ABB RAPID module: TaskModule.mod

MODULE TaskModule
    !*****************************************************
    !Module Name: TaskModule
    !Version:     1.0
    !Description: This module stroes ths data which are not shared among other tasks
    !Date:        2018-8-10
    !Author:      Michael
    !*****************************************************

    VAR num numStation:=1;
    VAR partdata pdTmpChk;
    VAR string sPartDataName;

    CONST num numPedestalBottomWidth:=100;
    CONST num numPedestalBottomHeight:=505;
    CONST num numPedestalAngle:=90;
    PERS num numPedestalVertexHeight:=455;

    VAR syncident SyncPositionerHomed;
    VAR syncident SyncWobjScanning;
    VAR syncident SyncWobjBranchScaning;
    VAR syncident SyncWobjBranchScaned;
    VAR syncident SyncWobjHeaderScaning;
    VAR syncident SyncWobjHeaderScaned;
    VAR syncident SyncWobjBranchScaningV2;
    VAR syncident SyncWobjBranchScanedV2;
    VAR syncident SyncWobjHeaderScaningV2;
    VAR syncident SyncWobjHeaderScanedV2;
    VAR syncident SyncWobjScaned;
    VAR syncident SyncBranchPeripherySmarTac;
    VAR syncident SyncHeaderPeripherySmarTac;
    VAR syncident SyncWobjRevised;

    VAR syncident SyncPositionerWeldApproached;
    VAR syncident SyncRobotsWeldApproached;
    VAR syncident SyncAllRobotsWeldStart;
    VAR syncident SyncAllRobotsWeldEnd;
    VAR syncident SyncRobotsWeldDeparted;

    VAR syncident SyncMoveLSubstituted1;
    VAR syncident SyncMoveLSubstituted2;

    VAR syncident SyncRobotsForTest11;
    VAR syncident SyncRobotsForTest12;
    VAR syncident SyncRobotsForTest13;

    VAR syncident SyncRobotsForTest21;
    VAR syncident SyncRobotsForTest22;
    VAR syncident SyncRobotsForTest23;
    VAR syncident SyncRobotsForTest24;
    VAR syncident SyncRobotsForTest25;
    VAR syncident SyncRobotsForTest26;

    VAR syncident SyncVerifyTrackHorizontal1;
    VAR syncident SyncVerifyTrackHorizontal2;
    VAR syncident SyncVerifyTrackHorizontal3;
    VAR syncident SyncVerifyTrackHorizontal4;
    VAR syncident SyncVerifyTrackHorizontal5;
    VAR syncident SyncVerifyTrackHorizontal6;
    VAR syncident SyncVerifyTrackHorizontal7;
    VAR syncident SyncVerifyTrackHorizontal8;

    VAR string strCurTaskName:="T_ROB1";
    VAR num numCurTaskNo:=1;
    VAR num numRobLayerCurTotal;
    VAR RECORDWeldTarget rRobLayerCur{30};
    VAR RECORDLayerParamter rLayerParamterCur;

    TASK PERS tooldata toolWeldGun:=[TRUE,[[80.8801,-0.792657,372.832],[0.950301,0.00218631,0.311128,-0.0110736]],[5.2,[34.6,-12.3,73.3],[1,0,0,0],0.048,0.077,0.012]];
    TASK PERS tooldata toolLaser:=[TRUE,[[-54.9581,16.2889,420.256],[0.999173,0.00179167,-0.00748378,0.0399198]],[5.2,[34.6,-12.3,73.3],[1,0,0,0],0.048,0.077,0.012]];
    TASK PERS extjoint extjointValue:=[4816.37,9E+09,9E+09,9E+09,9E+09,9E+09];

    TASK PERS robtarget robtApproachPlatoonSinking:=[[380,-200,190.17],[0.0294666,-0.614745,0.74898,0.245457],[-1,-1,0,1],[4837,9E+09,9E+09,9E+09,9E+09,9E+09]];
    TASK PERS robtarget robtDepartPlatoonSinking:=[[380,-200,190.17],[0.0294677,-0.614743,0.748982,0.245457],[-1,-1,0,1],[4837,9E+09,9E+09,9E+09,9E+09,9E+09]];

    TASK PERS robtarget robtApproachSaddle:=[[487.15,-501.33,347.1],[0.31599,-0.0842611,-0.937489,-0.119018],[-1,0,0,0],[4837,9E+09,9E+09,9E+09,9E+09,9E+09]];
    TASK PERS robtarget robtDepartSaddle:=[[487.15,-501.33,347.1],[0.315989,-0.0842597,-0.937489,-0.119018],[-1,0,0,0],[4837,9E+09,9E+09,9E+09,9E+09,9E+09]];

    TASK PERS robtarget robtApproachSaddleScan:=[[380,-301.92,219.63],[0.442137,-0.896947,4.32324E-05,3.41344E-05],[-1,-1,-1,1],[4837,9E+09,9E+09,9E+09,9E+09,9E+09]];
    TASK PERS robtarget robtDepartSaddleScan:=[[380,-301.92,219.64],[0.442138,-0.896947,4.317E-05,3.4008E-05],[-1,-1,-1,1],[4837,9E+09,9E+09,9E+09,9E+09,9E+09]];

    TASK PERS robtarget robtApproachPlatoonSinkingScan:=[[380,238.1,333.7],[0.270598,0.653281,-0.653282,0.270598],[0,0,1,1],[4837,9E+09,9E+09,9E+09,9E+09,9E+09]];
    TASK PERS robtarget robtDepartPlatoonSinkingScan:=[[380,238.1,333.7],[0.270598,0.653281,-0.653282,0.270598],[0,0,1,1],[4837,9E+09,9E+09,9E+09,9E+09,9E+09]];

    TASK PERS confdata confPlatoonSinkingOrigin:=[0,0,-1,1];
    TASK PERS confdata confSaddleOrigin:=[-1,0,-1,0];

    TASK PERS robtarget robtNext:=[[149.55,3.75943E-07,159.914],[0.348789,0.457656,-0.792683,-0.201373],[-1,0,-1,0],[4217,9E+09,9E+09,9E+09,9E+09,9E+09]];
    TASK PERS robtarget robtCircleEnd:=[[149.55,3.75943E-07,159.914],[0.348789,0.457656,-0.792683,-0.201373],[-1,1,-2,0],[4217,9E+09,9E+09,9E+09,9E+09,9E+09]];

    TASK PERS seamdata seamNext:=[0,0.5,[0,0,0,100,0,0,0,0,0],0,0,5,0,0,[0,0,1,140,0,0,0,0,0],0,1.5,[0,0,1,90,0,0,0,0,0],0.04,0,[0,0,0,0,0,0,0,0,0],0.5];
    TASK PERS welddata weldNext:=[7,0,[47,0,0,0,0,240,0,0,0],[0,0,0,0,0,0,0,0,0]];
    TASK PERS weavedata weaveNext:=[1,0,3.5,0,0,0,0,0,0,0,0,0,0,0,0];
    TASK PERS trackdata trackNext:=[0,FALSE,50,[0,0,0,0,0,0,0,0,0],[0,0,0,0,0,0,0]];
    TASK PERS adaptdata adaptNext:=[0,1,0,0,0.1,100,0.1,100];
    TASK PERS num numWeaveWidth90:=0;
    TASK PERS num numGrooveWidthNext:=0;

    VAR clock clockPartTimeConsume;
    TASK PERS num numTimeConsumeTotal:=623.885;

    !numTCSRotationX
    TASK PERS num numPlatoonSinkingPushDragAngle:=45;
    !numTCSRotationY
    TASK PERS num numPlatoonSinkingWorkAngle:=-10;

    TASK PERS jointtarget jointNext:=[[9E+09,9E+09,9E+09,9E+09,9E+09,9E+09],[0,66.4272,9E+09,9E+09,9E+09,9E+09]];
    TASK PERS speeddata speedLinearScan:=[19,500,5000,1000];

    TASK PERS string strWeldParametersLogFileName:="WeldParametersLog.csv";
    CONST string strWeldProcedureLogLogFileName:="WeldProcedureLog1.csv";

    CONST string strSSBLogFileName:="ScanSaddleBranch1.csv";
    CONST string strSSHLogFileName:="ScanSaddleHeader1.csv";

    !For saddle branch SmarTac
    TASK PERS num numSSBPointsTotal:=13;
    !Scan saddle branch range
    TASK PERS num numSSBAngleFrom:=225;
    TASK PERS num numSSBAngleTo:=330;

    !For saddle header SmarTac
    TASK PERS num numSSHPointsTotal:=13;
    !Scan saddle header range
    TASK PERS num numSSHAngleFrom:=180;
    TASK PERS num numSSHAngleTo:=90;

    !Scan saddle branch points
    TASK PERS robtarget robtSSBLaserSmarTacs{20}:=[[[339.589,-40.4111,208.15],[0.270598,0.270598,0.653282,0.653281],[0,0,0,1],[4837,9E+09,9E+09,9E+09,9E+09,9E+09]],[[346.207,-46.0883,208.15],[0.219975,0.219975,0.67202,0.67202],[0,0,0,1],[4837,9E+09,9E+09,9E+09,9E+09,9E+09]],[[353.611,-50.6927,208.15],[0.168069,0.168069,0.686843,0.686843],[0,0,0,1],[4837,9E+09,9E+09,9E+09,9E+09,9E+09]],[[361.63,-54.1171,208.15],[0.115184,0.115184,0.697662,0.697662],[0,0,0,1],[4837,9E+09,9E+09,9E+09,9E+09,9E+09]],[[370.076,-56.2818,208.15],[0.0616285,0.0616285,0.704416,0.704416],[0,0,0,1],[4837,9E+09,9E+09,9E+09,9E+09,9E+09]],[[378.753,-57.1364,208.15],[0.00771319,0.0077132,0.707065,0.707065],[0,0,1,1],[4837,9E+09,9E+09,9E+09,9E+09,9E+09]],[[387.46,-56.6611,208.15],[0.046247,0.046247,-0.705593,-0.705593],[-1,-1,1,1],[4837,9E+09,9E+09,9E+09,9E+09,9E+09]],[[395.992,-54.8668,208.15],[0.0999376,0.0999376,-0.700009,-0.700009],[-1,-1,1,1],[4837,9E+09,9E+09,9E+09,9E+09,9E+09]],[[404.153,-51.7955,208.15],[0.153046,0.153046,-0.690346,-0.690346],[-1,-1,1,1],[4837,9E+09,9E+09,9E+09,9E+09,9E+09]],[[411.751,-47.5185,208.15],[0.205262,0.205262,-0.676659,-0.676659],[-1,-1,1,1],[4837,9E+09,9E+09,9E+09,9E+09,9E+09]],[[418.61,-42.1354,208.15],[0.256282,0.256282,-0.659029,-0.659029],[-1,-1,1,1],[4837,9E+09,9E+09,9E+09,9E+09,9E+09]],[[424.57,-35.7715,208.15],[0.305809,0.305809,-0.637559,-0.637559],[-1,-1,1,1],[4837,9E+09,9E+09,9E+09,9E+09,9E+09]],[[429.493,-28.575,208.15],[0.353553,0.353553,-0.612372,-0.612372],[-1,-1,1,1],[4837,9E+09,9E+09,9E+09,9E+09,9E+09]],[[652.53,-493.33,1047.99],[0.459259,-0.544323,-0.447932,-0.54051],[-1,-1,1,1],[4837,9E+09,9E+09,9E+09,9E+09,9E+09]],[[652.53,-493.33,1047.99],[0.459259,-0.544323,-0.447932,-0.54051],[-1,0,-2,1],[4837,9E+09,9E+09,9E+09,9E+09,9E+09]],[[652.53,-493.33,1047.99],[0.459259,-0.544323,-0.447932,-0.54051],[-1,0,-2,1],[4837,9E+09,9E+09,9E+09,9E+09,9E+09]],[[652.53,-493.33,1047.99],[0.459259,-0.544323,-0.447932,-0.54051],[-1,0,-2,1],[4837,9E+09,9E+09,9E+09,9E+09,9E+09]],[[652.53,-493.33,1047.99],[0.459259,-0.544323,-0.447932,-0.54051],[-1,0,-2,1],[4837,9E+09,9E+09,9E+09,9E+09,9E+09]],[[652.53,-493.33,1047.99],[0.459259,-0.544323,-0.447932,-0.54051],[-1,0,-2,1],[4837,9E+09,9E+09,9E+09,9E+09,9E+09]],[[652.53,-493.33,1047.99],[0.459259,-0.544323,-0.447932,-0.54051],[-1,0,-2,1],[4837,9E+09,9E+09,9E+09,9E+09,9E+09]]];
    TASK PERS robtarget robtSSBWireSmarTacs{20}:=[[[428.493,28.575,188.15],[0.683013,0.183013,-0.683013,0.183013],[0,1,-3,1],[4838,9E+09,9E+09,9E+09,9E+09,9E+09]],[[422.779,36.7353,188.15],[0.664463,0.241845,-0.664463,0.241845],[0,1,-3,1],[4838,9E+09,9E+09,9E+09,9E+09,9E+09]],[[415.735,43.7794,188.15],[0.640856,0.298836,-0.640856,0.298836],[0,1,-3,1],[4838,9E+09,9E+09,9E+09,9E+09,9E+09]],[[407.575,49.4934,188.15],[0.612372,0.353553,-0.612372,0.353553],[0,0,-3,1],[4838,9E+09,9E+09,9E+09,9E+09,9E+09]],[[398.546,53.7034,188.15],[0.579228,0.40558,-0.579228,0.40558],[0,0,-3,1],[4838,9E+09,9E+09,9E+09,9E+09,9E+09]],[[388.924,56.2818,188.15],[0.541675,0.454519,-0.541675,0.454519],[0,0,-3,1],[4838,9E+09,9E+09,9E+09,9E+09,9E+09]],[[379,57.15,188.15],[0.5,0.5,-0.5,0.5],[0,0,-3,1],[4838,9E+09,9E+09,9E+09,9E+09,9E+09]],[[369.076,56.2818,188.15],[0.454519,0.541675,-0.454519,0.541675],[-1,-1,-2,1],[4838,9E+09,9E+09,9E+09,9E+09,9E+09]],[[359.454,53.7034,188.15],[0.40558,0.579228,-0.40558,0.579228],[-1,-1,-2,1],[4838,9E+09,9E+09,9E+09,9E+09,9E+09]],[[350.425,49.4934,188.15],[0.353553,0.612372,-0.353553,0.612372],[-1,-1,-2,1],[4838,9E+09,9E+09,9E+09,9E+09,9E+09]],[[342.265,43.7794,188.15],[0.298836,0.640856,-0.298836,0.640856],[-1,-2,-2,1],[4838,9E+09,9E+09,9E+09,9E+09,9E+09]],[[335.221,36.7353,188.15],[0.241845,0.664463,-0.241845,0.664463],[-1,-2,-2,1],[4838,9E+09,9E+09,9E+09,9E+09,9E+09]],[[329.507,28.575,188.15],[0.183013,0.683013,-0.183013,0.683013],[-1,-2,-2,1],[4838,9E+09,9E+09,9E+09,9E+09,9E+09]],[[652.53,-493.33,1047.99],[0.459259,-0.544323,-0.447932,-0.54051],[-1,-1,-2,1],[4837,9E+09,9E+09,9E+09,9E+09,9E+09]],[[652.53,-493.33,1047.99],[0.459259,-0.544323,-0.447932,-0.54051],[-1,0,-2,1],[4837,9E+09,9E+09,9E+09,9E+09,9E+09]],[[652.53,-493.33,1047.99],[0.459259,-0.544323,-0.447932,-0.54051],[-1,0,-2,1],[4837,9E+09,9E+09,9E+09,9E+09,9E+09]],[[652.53,-493.33,1047.99],[0.459259,-0.544323,-0.447932,-0.54051],[-1,0,-2,1],[4837,9E+09,9E+09,9E+09,9E+09,9E+09]],[[652.53,-493.33,1047.99],[0.459259,-0.544323,-0.447932,-0.54051],[-1,0,-2,1],[4837,9E+09,9E+09,9E+09,9E+09,9E+09]],[[652.53,-493.33,1047.99],[0.459259,-0.544323,-0.447932,-0.54051],[-1,0,-2,1],[4837,9E+09,9E+09,9E+09,9E+09,9E+09]],[[652.53,-493.33,1047.99],[0.459259,-0.544323,-0.447932,-0.54051],[-1,0,-2,1],[4837,9E+09,9E+09,9E+09,9E+09,9E+09]]];
    TASK PERS robtarget robtSSBLinerFrom:=[[427.815,-90,208.15],[3.09086E-08,3.09086E-08,-0.707107,-0.707107],[0,0,1,1],[4837,9E+09,9E+09,9E+09,9E+09,9E+09]];
    TASK PERS robtarget robtSSBLinerTo:=[[427.815,-90,208.15],[3.09086E-08,3.09086E-08,-0.707107,-0.707107],[0,0,1,1],[4837,9E+09,9E+09,9E+09,9E+09,9E+09]];

    !Scan saddle branch results, shared for all the four scan methods
    TASK PERS pose poseSSBs{20}:=[[[17.952,17.949,-0.0153198],[1,0,0,0]],[[1.39819,1.89476,-0.013504],[1,0,0,0]],[[1.19794,2.30891,-0.0127716],[1,0,0,0]],[[1.09225,3.15936,0.00701904],[1,0,0,0]],[[0.711761,4.05244,0.0107269],[1,0,0,0]],[[0.0821533,3.84193,-0.0236664],[1,0,0,0]],[[-0.370331,2.84446,0.0133057],[1,0,0,0]],[[-0.622101,2.14712,0.00906372],[1,0,0,0]],[[-1.77264,3.79015,0.0375366],[1,0,0,0]],[[-2.026,3.00191,-0.0130768],[1,0,0,0]],[[-5.25485,5.71828,0.0316315],[1,0,0,0]],[[-2.63602,2.12254,-0.0143127],[1,0,0,0]],[[-2.9296,1.71353,0.0193481],[1,0,0,0]],[[0,0,0],[1,0,0,0]],[[0,0,0],[1,0,0,0]],[[0,0,0],[1,0,0,0]],[[0,0,0],[1,0,0,0]],[[0,0,0],[1,0,0,0]],[[0,0,0],[1,0,0,0]],[[0,0,0],[1,0,0,0]]];
    TASK PERS num numSSBLaserValues{100}:=[0,0,0,0,0,0,0,0,0,0,0,0,0,0,0,0,0,0,0,0,0,0,0,0,0,0,0,0,0,0,0,0,0,0,0,0,0,0,0,0,0,0,0,0,0,0,0,0,0,0,0,0,0,0,0,0,0,0,0,0,0,0,0,0,0,0,0,0,0,0,0,0,0,0,0,0,0,0,0,0,0,0,0,0,0,0,0,0,0,0,0,0,0,0,0,0,0,0,0,0];
    TASK PERS robtarget robtSSBPeripherys{100}:=[[[920.345,-94.6578,259.235],[0.270602,0.270593,0.653289,0.653275],[0,0,0,1],[4202,9E+09,9E+09,9E+09,9E+09,9E+09]],[[347.605,-44.1936,208.136],[0.219979,0.219977,0.672024,0.672014],[0,0,0,1],[4837,9E+09,9E+09,9E+09,9E+09,9E+09]],[[354.809,-48.3838,208.137],[0.168074,0.168066,0.686843,0.686841],[0,0,0,1],[4837,9E+09,9E+09,9E+09,9E+09,9E+09]],[[362.722,-50.9577,208.157],[0.115179,0.115206,0.697653,0.697669],[0,0,0,1],[4837,9E+09,9E+09,9E+09,9E+09,9E+09]],[[370.788,-52.2293,208.161],[0.0616358,0.0616132,0.704405,0.704427],[0,0,0,1],[4837,9E+09,9E+09,9E+09,9E+09,9E+09]],[[378.835,-53.2945,208.126],[0.00771569,0.00771062,0.707077,0.707053],[0,0,1,1],[4837,9E+09,9E+09,9E+09,9E+09,9E+09]],[[387.089,-53.8166,208.163],[0.0462415,0.0462523,-0.705592,-0.705594],[-1,-1,1,1],[4837,9E+09,9E+09,9E+09,9E+09,9E+09]],[[395.37,-52.7197,208.159],[0.0999338,0.0999283,-0.700005,-0.700014],[-1,-1,1,1],[4837,9E+09,9E+09,9E+09,9E+09,9E+09]],[[402.38,-48.0053,208.188],[0.153049,0.153049,-0.690324,-0.690366],[-1,-1,1,1],[4837,9E+09,9E+09,9E+09,9E+09,9E+09]],[[409.725,-44.5166,208.137],[0.205273,0.20527,-0.676661,-0.676652],[-1,-1,1,1],[4837,9E+09,9E+09,9E+09,9E+09,9E+09]],[[413.355,-36.4171,208.182],[0.256285,0.256298,-0.659006,-0.659045],[-1,-1,1,1],[4837,9E+09,9E+09,9E+09,9E+09,9E+09]],[[421.934,-33.649,208.136],[0.305815,0.3058,-0.637569,-0.637549],[-1,-1,1,1],[4837,9E+09,9E+09,9E+09,9E+09,9E+09]],[[426.564,-26.8615,208.169],[0.353544,0.353553,-0.612368,-0.612383],[-1,-1,1,1],[4837,9E+09,9E+09,9E+09,9E+09,9E+09]],[[75.54,-110.49,75.53],[0.104911,-0.592891,0.59209,0.535634],[-1,-2,0,1],[3747.5,9E+09,9E+09,9E+09,9E+09,9E+09]],[[75.54,-110.49,75.53],[0.104911,-0.592891,0.59209,0.535634],[-1,0,-1,0],[3747.5,9E+09,9E+09,9E+09,9E+09,9E+09]],[[75.54,-110.49,75.53],[0.104911,-0.592891,0.59209,0.535634],[-1,0,-1,0],[3747.5,9E+09,9E+09,9E+09,9E+09,9E+09]],[[75.54,-110.49,75.53],[0.104911,-0.592891,0.59209,0.535634],[-1,0,-1,0],[3747.5,9E+09,9E+09,9E+09,9E+09,9E+09]],[[75.54,-110.49,75.53],[0.104911,-0.592891,0.59209,0.535634],[-1,0,-1,0],[3747.5,9E+09,9E+09,9E+09,9E+09,9E+09]],[[75.54,-110.49,75.53],[0.104911,-0.592891,0.59209,0.535634],[-1,0,-1,0],[3747.5,9E+09,9E+09,9E+09,9E+09,9E+09]],[[75.54,-110.49,75.53],[0.104911,-0.592891,0.59209,0.535634],[-1,0,-1,0],[3747.5,9E+09,9E+09,9E+09,9E+09,9E+09]],[[75.54,-110.49,75.53],[0.104911,-0.592891,0.59209,0.535634],[-1,0,-1,0],[3747.5,9E+09,9E+09,9E+09,9E+09,9E+09]],[[75.54,-110.49,75.53],[0.104911,-0.592891,0.59209,0.535634],[-1,0,-1,0],[3747.5,9E+09,9E+09,9E+09,9E+09,9E+09]],[[75.54,-110.49,75.53],[0.104911,-0.592891,0.59209,0.535634],[-1,0,-1,0],[3747.5,9E+09,9E+09,9E+09,9E+09,9E+09]],[[75.54,-110.49,75.53],[0.104911,-0.592891,0.59209,0.535634],[-1,0,-1,0],[3747.5,9E+09,9E+09,9E+09,9E+09,9E+09]],[[75.54,-110.49,75.53],[0.104911,-0.592891,0.59209,0.535634],[-1,0,-1,0],[3747.5,9E+09,9E+09,9E+09,9E+09,9E+09]],[[75.54,-110.49,75.53],[0.104911,-0.592891,0.59209,0.535634],[-1,0,-1,0],[3747.5,9E+09,9E+09,9E+09,9E+09,9E+09]],[[75.54,-110.49,75.53],[0.104911,-0.592891,0.59209,0.535634],[-1,0,-1,0],[3747.5,9E+09,9E+09,9E+09,9E+09,9E+09]],[[75.54,-110.49,75.53],[0.104911,-0.592891,0.59209,0.535634],[-1,0,-1,0],[3747.5,9E+09,9E+09,9E+09,9E+09,9E+09]],[[75.54,-110.49,75.53],[0.104911,-0.592891,0.59209,0.535634],[-1,0,-1,0],[3747.5,9E+09,9E+09,9E+09,9E+09,9E+09]],[[75.54,-110.49,75.53],[0.104911,-0.592891,0.59209,0.535634],[-1,0,-1,0],[3747.5,9E+09,9E+09,9E+09,9E+09,9E+09]],[[75.54,-110.49,75.53],[0.104911,-0.592891,0.59209,0.535634],[-1,0,-1,0],[3747.5,9E+09,9E+09,9E+09,9E+09,9E+09]],[[75.54,-110.49,75.53],[0.104911,-0.592891,0.59209,0.535634],[-1,0,-1,0],[3747.5,9E+09,9E+09,9E+09,9E+09,9E+09]],[[75.54,-110.49,75.53],[0.104911,-0.592891,0.59209,0.535634],[-1,0,-1,0],[3747.5,9E+09,9E+09,9E+09,9E+09,9E+09]],[[75.54,-110.49,75.53],[0.104911,-0.592891,0.59209,0.535634],[-1,0,-1,0],[3747.5,9E+09,9E+09,9E+09,9E+09,9E+09]],[[75.54,-110.49,75.53],[0.104911,-0.592891,0.59209,0.535634],[-1,0,-1,0],[3747.5,9E+09,9E+09,9E+09,9E+09,9E+09]],[[75.54,-110.49,75.53],[0.104911,-0.592891,0.59209,0.535634],[-1,0,-1,0],[3747.5,9E+09,9E+09,9E+09,9E+09,9E+09]],[[75.54,-110.49,75.53],[0.104911,-0.592891,0.59209,0.535634],[-1,0,-1,0],[3747.5,9E+09,9E+09,9E+09,9E+09,9E+09]],[[75.54,-110.49,75.53],[0.104911,-0.592891,0.59209,0.535634],[-1,0,-1,0],[3747.5,9E+09,9E+09,9E+09,9E+09,9E+09]],[[75.54,-110.49,75.53],[0.104911,-0.592891,0.59209,0.535634],[-1,0,-1,0],[3747.5,9E+09,9E+09,9E+09,9E+09,9E+09]],[[75.54,-110.49,75.53],[0.104911,-0.592891,0.59209,0.535634],[-1,0,-1,0],[3747.5,9E+09,9E+09,9E+09,9E+09,9E+09]],[[75.54,-110.49,75.53],[0.104911,-0.592891,0.59209,0.535634],[-1,0,-1,0],[3747.5,9E+09,9E+09,9E+09,9E+09,9E+09]],[[75.54,-110.49,75.53],[0.104911,-0.592891,0.59209,0.535634],[-1,0,-1,0],[3747.5,9E+09,9E+09,9E+09,9E+09,9E+09]],[[75.54,-110.49,75.53],[0.104911,-0.592891,0.59209,0.535634],[-1,0,-1,0],[3747.5,9E+09,9E+09,9E+09,9E+09,9E+09]],[[75.54,-110.49,75.53],[0.104911,-0.592891,0.59209,0.535634],[-1,0,-1,0],[3747.5,9E+09,9E+09,9E+09,9E+09,9E+09]],[[75.54,-110.49,75.53],[0.104911,-0.592891,0.59209,0.535634],[-1,0,-1,0],[3747.5,9E+09,9E+09,9E+09,9E+09,9E+09]],[[75.54,-110.49,75.53],[0.104911,-0.592891,0.59209,0.535634],[-1,0,-1,0],[3747.5,9E+09,9E+09,9E+09,9E+09,9E+09]],[[75.54,-110.49,75.53],[0.104911,-0.592891,0.59209,0.535634],[-1,0,-1,0],[3747.5,9E+09,9E+09,9E+09,9E+09,9E+09]],[[75.54,-110.49,75.53],[0.104911,-0.592891,0.59209,0.535634],[-1,0,-1,0],[3747.5,9E+09,9E+09,9E+09,9E+09,9E+09]],[[75.54,-110.49,75.53],[0.104911,-0.592891,0.59209,0.535634],[-1,0,-1,0],[3747.5,9E+09,9E+09,9E+09,9E+09,9E+09]],[[75.54,-110.49,75.53],[0.104911,-0.592891,0.59209,0.535634],[-1,0,-1,0],[3747.5,9E+09,9E+09,9E+09,9E+09,9E+09]],[[75.54,-110.49,75.53],[0.104911,-0.592891,0.59209,0.535634],[-1,0,-1,0],[3747.5,9E+09,9E+09,9E+09,9E+09,9E+09]],[[75.54,-110.49,75.53],[0.104911,-0.592891,0.59209,0.535634],[-1,0,-1,0],[3747.5,9E+09,9E+09,9E+09,9E+09,9E+09]],[[75.54,-110.49,75.53],[0.104911,-0.592891,0.59209,0.535634],[-1,0,-1,0],[3747.5,9E+09,9E+09,9E+09,9E+09,9E+09]],[[75.54,-110.49,75.53],[0.104911,-0.592891,0.59209,0.535634],[-1,0,-1,0],[3747.5,9E+09,9E+09,9E+09,9E+09,9E+09]],[[75.54,-110.49,75.53],[0.104911,-0.592891,0.59209,0.535634],[-1,0,-1,0],[3747.5,9E+09,9E+09,9E+09,9E+09,9E+09]],[[75.54,-110.49,75.53],[0.104911,-0.592891,0.59209,0.535634],[-1,0,-1,0],[3747.5,9E+09,9E+09,9E+09,9E+09,9E+09]],[[75.54,-110.49,75.53],[0.104911,-0.592891,0.59209,0.535634],[-1,0,-1,0],[3747.5,9E+09,9E+09,9E+09,9E+09,9E+09]],[[75.54,-110.49,75.53],[0.104911,-0.592891,0.59209,0.535634],[-1,0,-1,0],[3747.5,9E+09,9E+09,9E+09,9E+09,9E+09]],[[75.54,-110.49,75.53],[0.104911,-0.592891,0.59209,0.535634],[-1,0,-1,0],[3747.5,9E+09,9E+09,9E+09,9E+09,9E+09]],[[75.54,-110.49,75.53],[0.104911,-0.592891,0.59209,0.535634],[-1,0,-1,0],[3747.5,9E+09,9E+09,9E+09,9E+09,9E+09]],[[75.54,-110.49,75.53],[0.104911,-0.592891,0.59209,0.535634],[-1,0,-1,0],[3747.5,9E+09,9E+09,9E+09,9E+09,9E+09]],[[75.54,-110.49,75.53],[0.104911,-0.592891,0.59209,0.535634],[-1,0,-1,0],[3747.5,9E+09,9E+09,9E+09,9E+09,9E+09]],[[75.54,-110.49,75.53],[0.104911,-0.592891,0.59209,0.535634],[-1,0,-1,0],[3747.5,9E+09,9E+09,9E+09,9E+09,9E+09]],[[75.54,-110.49,75.53],[0.104911,-0.592891,0.59209,0.535634],[-1,0,-1,0],[3747.5,9E+09,9E+09,9E+09,9E+09,9E+09]],[[75.54,-110.49,75.53],[0.104911,-0.592891,0.59209,0.535634],[-1,0,-1,0],[3747.5,9E+09,9E+09,9E+09,9E+09,9E+09]],[[75.54,-110.49,75.53],[0.104911,-0.592891,0.59209,0.535634],[-1,0,-1,0],[3747.5,9E+09,9E+09,9E+09,9E+09,9E+09]],[[75.54,-110.49,75.53],[0.104911,-0.592891,0.59209,0.535634],[-1,0,-1,0],[3747.5,9E+09,9E+09,9E+09,9E+09,9E+09]],[[75.54,-110.49,75.53],[0.104911,-0.592891,0.59209,0.535634],[-1,0,-1,0],[3747.5,9E+09,9E+09,9E+09,9E+09,9E+09]],[[75.54,-110.49,75.53],[0.104911,-0.592891,0.59209,0.535634],[-1,0,-1,0],[3747.5,9E+09,9E+09,9E+09,9E+09,9E+09]],[[75.54,-110.49,75.53],[0.104911,-0.592891,0.59209,0.535634],[-1,0,-1,0],[3747.5,9E+09,9E+09,9E+09,9E+09,9E+09]],[[75.54,-110.49,75.53],[0.104911,-0.592891,0.59209,0.535634],[-1,0,-1,0],[3747.5,9E+09,9E+09,9E+09,9E+09,9E+09]],[[75.54,-110.49,75.53],[0.104911,-0.592891,0.59209,0.535634],[-1,0,-1,0],[3747.5,9E+09,9E+09,9E+09,9E+09,9E+09]],[[75.54,-110.49,75.53],[0.104911,-0.592891,0.59209,0.535634],[-1,0,-1,0],[3747.5,9E+09,9E+09,9E+09,9E+09,9E+09]],[[75.54,-110.49,75.53],[0.104911,-0.592891,0.59209,0.535634],[-1,0,-1,0],[3747.5,9E+09,9E+09,9E+09,9E+09,9E+09]],[[75.54,-110.49,75.53],[0.104911,-0.592891,0.59209,0.535634],[-1,0,-1,0],[3747.5,9E+09,9E+09,9E+09,9E+09,9E+09]],[[75.54,-110.49,75.53],[0.104911,-0.592891,0.59209,0.535634],[-1,0,-1,0],[3747.5,9E+09,9E+09,9E+09,9E+09,9E+09]],[[75.54,-110.49,75.53],[0.104911,-0.592891,0.59209,0.535634],[-1,0,-1,0],[3747.5,9E+09,9E+09,9E+09,9E+09,9E+09]],[[75.54,-110.49,75.53],[0.104911,-0.592891,0.59209,0.535634],[-1,0,-1,0],[3747.5,9E+09,9E+09,9E+09,9E+09,9E+09]],[[75.54,-110.49,75.53],[0.104911,-0.592891,0.59209,0.535634],[-1,0,-1,0],[3747.5,9E+09,9E+09,9E+09,9E+09,9E+09]],[[75.54,-110.49,75.53],[0.104911,-0.592891,0.59209,0.535634],[-1,0,-1,0],[3747.5,9E+09,9E+09,9E+09,9E+09,9E+09]],[[75.54,-110.49,75.53],[0.104911,-0.592891,0.59209,0.535634],[-1,0,-1,0],[3747.5,9E+09,9E+09,9E+09,9E+09,9E+09]],[[75.54,-110.49,75.53],[0.104911,-0.592891,0.59209,0.535634],[-1,0,-1,0],[3747.5,9E+09,9E+09,9E+09,9E+09,9E+09]],[[75.54,-110.49,75.53],[0.104911,-0.592891,0.59209,0.535634],[-1,0,-1,0],[3747.5,9E+09,9E+09,9E+09,9E+09,9E+09]],[[75.54,-110.49,75.53],[0.104911,-0.592891,0.59209,0.535634],[-1,0,-1,0],[3747.5,9E+09,9E+09,9E+09,9E+09,9E+09]],[[75.54,-110.49,75.53],[0.104911,-0.592891,0.59209,0.535634],[-1,0,-1,0],[3747.5,9E+09,9E+09,9E+09,9E+09,9E+09]],[[75.54,-110.49,75.53],[0.104911,-0.592891,0.59209,0.535634],[-1,0,-1,0],[3747.5,9E+09,9E+09,9E+09,9E+09,9E+09]],[[75.54,-110.49,75.53],[0.104911,-0.592891,0.59209,0.535634],[-1,0,-1,0],[3747.5,9E+09,9E+09,9E+09,9E+09,9E+09]],[[75.54,-110.49,75.53],[0.104911,-0.592891,0.59209,0.535634],[-1,0,-1,0],[3747.5,9E+09,9E+09,9E+09,9E+09,9E+09]],[[75.54,-110.49,75.53],[0.104911,-0.592891,0.59209,0.535634],[-1,0,-1,0],[3747.5,9E+09,9E+09,9E+09,9E+09,9E+09]],[[75.54,-110.49,75.53],[0.104911,-0.592891,0.59209,0.535634],[-1,0,-1,0],[3747.5,9E+09,9E+09,9E+09,9E+09,9E+09]],[[75.54,-110.49,75.53],[0.104911,-0.592891,0.59209,0.535634],[-1,0,-1,0],[3747.5,9E+09,9E+09,9E+09,9E+09,9E+09]],[[75.54,-110.49,75.53],[0.104911,-0.592891,0.59209,0.535634],[-1,0,-1,0],[3747.5,9E+09,9E+09,9E+09,9E+09,9E+09]],[[75.54,-110.49,75.53],[0.104911,-0.592891,0.59209,0.535634],[-1,0,-1,0],[3747.5,9E+09,9E+09,9E+09,9E+09,9E+09]],[[75.54,-110.49,75.53],[0.104911,-0.592891,0.59209,0.535634],[-1,0,-1,0],[3747.5,9E+09,9E+09,9E+09,9E+09,9E+09]],[[75.54,-110.49,75.53],[0.104911,-0.592891,0.59209,0.535634],[-1,0,-1,0],[3747.5,9E+09,9E+09,9E+09,9E+09,9E+09]],[[75.54,-110.49,75.53],[0.104911,-0.592891,0.59209,0.535634],[-1,0,-1,0],[3747.5,9E+09,9E+09,9E+09,9E+09,9E+09]],[[75.54,-110.49,75.53],[0.104911,-0.592891,0.59209,0.535634],[-1,0,-1,0],[3747.5,9E+09,9E+09,9E+09,9E+09,9E+09]],[[75.54,-110.49,75.53],[0.104911,-0.592891,0.59209,0.535634],[-1,0,-1,0],[3747.5,9E+09,9E+09,9E+09,9E+09,9E+09]],[[75.54,-110.49,75.53],[0.104911,-0.592891,0.59209,0.535634],[-1,0,-1,0],[3747.5,9E+09,9E+09,9E+09,9E+09,9E+09]],[[75.54,-110.49,75.53],[0.104911,-0.592891,0.59209,0.535634],[-1,0,-1,0],[3747.5,9E+09,9E+09,9E+09,9E+09,9E+09]]];
    TASK PERS pos posSSBPeripherys{100}:=[[920.345,-94.6578,259.235],[347.605,-44.1936,208.136],[354.809,-48.3838,208.137],[362.722,-50.9577,208.157],[370.788,-52.2293,208.161],[378.835,-53.2945,208.126],[387.089,-53.8166,208.163],[395.37,-52.7197,208.159],[402.38,-48.0053,208.188],[409.725,-44.5166,208.137],[413.355,-36.4171,208.182],[421.934,-33.649,208.136],[426.564,-26.8615,208.169],[403.721,-54.5007,218.144],[402.695,-54.7914,218.15],[401.613,-55.2287,218.151],[400.612,-55.6663,218.16],[399.584,-55.6652,218.161],[398.506,-55.6653,218.154],[397.454,-56.5454,218.153],[396.435,-56.5484,218.147],[395.393,-57.1338,218.149],[394.377,-57.573,218.149],[393.302,-57.5728,218.152],[392.269,-57.8653,218.151],[391.229,-58.0135,218.151],[390.146,-58.0121,218.15],[389.116,-58.1615,218.148],[388.11,-58.601,218.152],[387.028,-58.5999,218.152],[386,-58.6,218.154],[384.982,-58.6014,218.153],[383.916,-58.4571,218.152],[382.868,-58.6069,218.153],[381.835,-58.4659,218.153],[380.789,-58.1789,218.151],[379.733,-58.1848,218.151],[378.699,-58.6326,218.147],[377.665,-58.489,218.152],[376.646,-58.486,218.161],[375.577,-58.6304,218.172],[374.516,-57.3071,218.178],[373.483,-57.5924,218.186],[372.468,-58.4606,218.198],[371.413,-56.8386,218.212],[370.378,-57.1252,218.221],[369.332,-56.8308,218.22],[368.287,-57.1221,218.223],[367.205,-56.5413,218.213],[366.179,-55.6646,218.209],[365.152,-55.668,218.196],[364.087,-55.0838,218.188],[363.017,-55.232,218.18],[361.985,-54.7921,218.174],[360.946,-54.4989,218.172],[359.89,-53.7688,218.165],[358.836,-54.0598,218.167],[357.811,-53.3263,218.165],[356.755,-52.301,218.162],[355.671,-51.7184,218.156],[354.682,-51.1319,218.154],[353.654,-50.5491,218.148],[352.593,-50.4035,218.147],[351.534,-50.1095,218.146],[350.499,-49.3779,218.145],[349.454,-48.3511,218.147],[348.381,-47.3241,218.148],[347.337,-46.5856,218.152],[346.328,-45.9985,218.158],[345.319,-44.9732,218.159],[344.243,-44.0985,218.151],[343.187,-42.9305,218.149],[342.157,-42.7851,218.144],[341.097,-41.4677,218.145],[340.046,-40.0006,218.147],[339.014,-39.9967,218.153],[337.969,-39.9951,218.152],[336.914,-39.9978,218.148],[335.866,-40,218.144],[334.859,-40.003,218.141],[344.243,-44.0985,218.151],[343.187,-42.9305,218.149],[342.157,-42.7851,218.144],[341.097,-41.4677,218.145],[340.046,-40.0006,218.147],[339.014,-39.9967,218.153],[337.969,-39.9951,218.152],[336.914,-39.9978,218.148],[335.866,-40,218.144],[334.859,-40.003,218.141],[332.054,-39.994,188.152],[0,0,0],[0,0,0],[0,0,0],[0,0,0],[0,0,0],[0,0,0],[0,0,0],[0,0,0],[0,0,0]];
    TASK PERS robtarget robtSSBPeripheryCenter:=[[378.584,-53.7077,158.208],[5.69172E-06,-1.40379E-06,-0.70708,-0.707133],[0,-1,1,1],[4837,9E+09,9E+09,9E+09,9E+09,9E+09]];
    TASK PERS pose poseSSBPeripheryCenter:=[[-0.00570679,3.44234,0.0576935],[1,0,0,0]];

    !Scan saddle header points
    TASK PERS robtarget robtSSHLaserSmarTacs{20}:=[[[1129.25,-159.25,-1.39221E-05],[0.707107,-0.707107,0,0],[-1,-1,-1,1],[4262,9E+09,9E+09,9E+09,9E+09,9E+09]],[[1129.25,-157.888,20.7863],[0.659346,-0.75184,0,0],[-1,-1,-1,1],[4262,9E+09,9E+09,9E+09,9E+09,9E+09]],[[1129.25,-153.824,41.2169],[0.608761,-0.793353,0,0],[-1,-1,-1,1],[4262,9E+09,9E+09,9E+09,9E+09,9E+09]],[[1129.25,-147.128,60.9423],[0.55557,-0.83147,0,0],[-1,-1,-1,1],[4262,9E+09,9E+09,9E+09,9E+09,9E+09]],[[1129.25,-137.915,79.625],[0.5,-0.866025,0,0],[-1,-1,-1,1],[4262,9E+09,9E+09,9E+09,9E+09,9E+09]],[[1129.25,-126.342,96.9453],[0.442289,-0.896873,0,0],[-1,-1,-1,1],[4262,9E+09,9E+09,9E+09,9E+09,9E+09]],[[1129.25,-112.607,112.607],[0.382683,-0.92388,0,0],[-1,-1,-1,1],[4262,9E+09,9E+09,9E+09,9E+09,9E+09]],[[1129.25,-96.9453,126.342],[0.321439,-0.94693,0,0],[-1,-1,-1,1],[4262,9E+09,9E+09,9E+09,9E+09,9E+09]],[[1129.25,-79.625,137.915],[0.258819,-0.965926,0,0],[-1,0,-2,0],[4262,9E+09,9E+09,9E+09,9E+09,9E+09]],[[1129.25,-60.9423,147.128],[0.19509,-0.980785,0,0],[-1,0,-2,0],[4262,9E+09,9E+09,9E+09,9E+09,9E+09]],[[1129.25,-41.2169,153.824],[0.130526,-0.991445,0,0],[-1,0,-2,0],[4262,9E+09,9E+09,9E+09,9E+09,9E+09]],[[1129.25,-20.7863,157.888],[0.0654032,-0.997859,0,0],[-1,0,-2,0],[4262,9E+09,9E+09,9E+09,9E+09,9E+09]],[[1129.25,-6.96104E-06,159.25],[4.37114E-08,1,0,0],[-1,0,-2,0],[4262,9E+09,9E+09,9E+09,9E+09,9E+09]],[[652.53,-493.33,1047.99],[0.459259,-0.544323,-0.447932,-0.54051],[-1,0,-2,0],[4837,9E+09,9E+09,9E+09,9E+09,9E+09]],[[652.53,-493.33,1047.99],[0.459259,-0.544323,-0.447932,-0.54051],[-1,0,-2,1],[4837,9E+09,9E+09,9E+09,9E+09,9E+09]],[[652.53,-493.33,1047.99],[0.459259,-0.544323,-0.447932,-0.54051],[-1,0,-2,1],[4837,9E+09,9E+09,9E+09,9E+09,9E+09]],[[652.53,-493.33,1047.99],[0.459259,-0.544323,-0.447932,-0.54051],[-1,0,-2,1],[4837,9E+09,9E+09,9E+09,9E+09,9E+09]],[[652.53,-493.33,1047.99],[0.459259,-0.544323,-0.447932,-0.54051],[-1,0,-2,1],[4837,9E+09,9E+09,9E+09,9E+09,9E+09]],[[652.53,-493.33,1047.99],[0.459259,-0.544323,-0.447932,-0.54051],[-1,0,-2,1],[4837,9E+09,9E+09,9E+09,9E+09,9E+09]],[[652.53,-493.33,1047.99],[0.459259,-0.544323,-0.447932,-0.54051],[-1,0,-2,1],[4837,9E+09,9E+09,9E+09,9E+09,9E+09]]];
    TASK PERS robtarget robtSSHWireSmarTacs{20}:=[[[296.85,108.15,0],[0.5,0.5,-0.5,0.5],[-1,-1,2,1],[4838,9E+09,9E+09,9E+09,9E+09,9E+09]],[[296.85,107.225,14.1164],[0.466228,0.531631,-0.531631,0.466228],[-1,-1,2,1],[4838,9E+09,9E+09,9E+09,9E+09,9E+09]],[[296.85,104.465,27.9913],[0.430459,0.560986,-0.560986,0.430459],[-1,-1,2,1],[4838,9E+09,9E+09,9E+09,9E+09,9E+09]],[[296.85,99.9176,41.3872],[0.392847,0.587938,-0.587938,0.392848],[-1,0,1,0],[4838,9E+09,9E+09,9E+09,9E+09,9E+09]],[[296.85,93.6606,54.075],[0.353553,0.612372,-0.612372,0.353553],[-1,0,1,0],[4838,9E+09,9E+09,9E+09,9E+09,9E+09]],[[296.85,85.8012,65.8375],[0.312745,0.634185,-0.634185,0.312745],[-1,0,1,0],[4838,9E+09,9E+09,9E+09,9E+09,9E+09]],[[296.85,76.4736,76.4736],[0.270598,0.653282,0.653281,-0.270598],[-1,-1,0,1],[4838,9E+09,9E+09,9E+09,9E+09,9E+09]],[[296.85,65.8375,85.8012],[0.227292,0.669581,0.669581,-0.227292],[-1,-1,0,1],[4838,9E+09,9E+09,9E+09,9E+09,9E+09]],[[296.85,54.075,93.6607],[0.183013,0.683013,0.683013,-0.183013],[-1,-1,0,1],[4838,9E+09,9E+09,9E+09,9E+09,9E+09]],[[296.85,41.3872,99.9176],[0.13795,0.69352,0.69352,-0.13795],[-1,-1,0,1],[4838,9E+09,9E+09,9E+09,9E+09,9E+09]],[[296.85,27.9913,104.465],[0.092296,0.701057,0.701057,-0.092296],[-1,-1,0,1],[4838,9E+09,9E+09,9E+09,9E+09,9E+09]],[[296.85,14.1164,107.225],[0.046247,0.705593,0.705593,-0.046247],[-1,0,-1,0],[4838,9E+09,9E+09,9E+09,9E+09,9E+09]],[[296.85,-4.72739E-06,108.15],[3.09086E-08,-0.707107,-0.707107,-3.09086E-08],[-1,0,-1,0],[4838,9E+09,9E+09,9E+09,9E+09,9E+09]],[[652.53,-493.33,1047.99],[0.459259,-0.544323,-0.447932,-0.54051],[-1,0,-1,0],[4837,9E+09,9E+09,9E+09,9E+09,9E+09]],[[652.53,-493.33,1047.99],[0.459259,-0.544323,-0.447932,-0.54051],[-1,0,-2,1],[4837,9E+09,9E+09,9E+09,9E+09,9E+09]],[[652.53,-493.33,1047.99],[0.459259,-0.544323,-0.447932,-0.54051],[-1,0,-2,1],[4837,9E+09,9E+09,9E+09,9E+09,9E+09]],[[652.53,-493.33,1047.99],[0.459259,-0.544323,-0.447932,-0.54051],[-1,0,-2,1],[4837,9E+09,9E+09,9E+09,9E+09,9E+09]],[[652.53,-493.33,1047.99],[0.459259,-0.544323,-0.447932,-0.54051],[-1,0,-2,1],[4837,9E+09,9E+09,9E+09,9E+09,9E+09]],[[652.53,-493.33,1047.99],[0.459259,-0.544323,-0.447932,-0.54051],[-1,0,-2,1],[4837,9E+09,9E+09,9E+09,9E+09,9E+09]],[[652.53,-493.33,1047.99],[0.459259,-0.544323,-0.447932,-0.54051],[-1,0,-2,1],[4837,9E+09,9E+09,9E+09,9E+09,9E+09]]];
    TASK PERS robtarget robtSSHLinerFrom:=[[452.15,-78.15,88.5913],[0.5,-0.5,-0.5,-0.5],[-1,-1,-1,1],[4837,9E+09,9E+09,9E+09,9E+09,9E+09]];
    TASK PERS robtarget robtSSHLinerTo:=[[452.15,-78.15,-88.5913],[0.5,-0.5,-0.5,-0.5],[-1,-1,-1,1],[4837,9E+09,9E+09,9E+09,9E+09,9E+09]];

    !Scan saddle header results, shared for all the four scan methods
    TASK PERS pose poseSSHs{20}:=[[[-0.0262756,-1.74011,-0.0842074],[1,0,0,0]],[[0.00857544,-1.63525,-0.318074],[1,0,0,0]],[[-0.028656,-1.64377,-0.546583],[1,0,0,0]],[[0.0638428,-2.0858,-0.993671],[1,0,0,0]],[[0.0242615,-5.82465,-3.91956],[1,0,0,0]],[[-0.00445557,-2.85303,-2.25892],[1,0,0,0]],[[-0.0636902,-4.71622,-4.46343],[1,0,0,0]],[[-0.0174561,-1.48105,-1.78532],[1,0,0,0]],[[-0.0214844,-1.60992,-2.29945],[1,0,0,0]],[[-0.0274048,-2.24935,-4.57064],[1,0,0,0]],[[0.00231934,-0.64773,-2.24944],[1,0,0,0]],[[-0.0207214,-0.326895,-2.32129],[1,0,0,0]],[[-0.0108948,0.00979681,-3.05504],[1,0,0,0]],[[0,0,0],[1,0,0,0]],[[0,0,0],[1,0,0,0]],[[0,0,0],[1,0,0,0]],[[0,0,0],[1,0,0,0]],[[0,0,0],[1,0,0,0]],[[0,0,0],[1,0,0,0]],[[0,0,0],[1,0,0,0]]];
    TASK PERS num numSSHLaserValues{100}:=[0,0,0,0,0,0,0,0,0,0,0,0,0,0,0,0,0,0,0,0,0,0,0,0,0,0,0,0,0,0,0,0,0,0,0,0,0,0,0,0,0,0,0,0,0,0,0,0,0,0,0,0,0,0,0,0,0,0,0,0,0,0,0,0,0,0,0,0,0,0,0,0,0,0,0,0,0,0,0,0,0,0,0,0,0,0,0,0,0,0,0,0,0,0,0,0,0,0,0,0];
    TASK PERS robtarget robtSSHPeripherys{100}:=[[[296.824,106.41,-0.0842074],[0.499958,0.500028,-0.500074,0.49994],[-1,-1,2,1],[4838,9E+09,9E+09,9E+09,9E+09,9E+09]],[[296.859,105.59,13.7983],[0.466186,0.531648,-0.531681,0.466194],[-1,-1,2,1],[4838,9E+09,9E+09,9E+09,9E+09,9E+09]],[[296.821,102.821,27.4447],[0.430412,0.561012,-0.561049,0.430389],[-1,-1,2,1],[4838,9E+09,9E+09,9E+09,9E+09,9E+09]],[[296.914,97.8318,40.3935],[0.392741,0.587978,-0.587986,0.392822],[-1,0,1,0],[4838,9E+09,9E+09,9E+09,9E+09,9E+09]],[[296.874,87.836,50.1554],[0.353284,0.612457,-0.612578,0.353322],[-1,0,1,0],[4838,9E+09,9E+09,9E+09,9E+09,9E+09]],[[296.846,82.9481,63.5786],[0.312722,0.634193,-0.634199,0.312722],[-1,0,1,0],[4838,9E+09,9E+09,9E+09,9E+09,9E+09]],[[296.786,71.7574,72.0102],[0.270652,0.653251,0.653232,-0.270739],[-1,-1,0,1],[4838,9E+09,9E+09,9E+09,9E+09,9E+09]],[[296.833,64.3565,84.0158],[0.227343,0.669554,0.669563,-0.227371],[-1,-1,0,1],[4838,9E+09,9E+09,9E+09,9E+09,9E+09]],[[296.829,52.4651,91.3612],[0.183138,0.682977,0.682975,-0.183162],[-1,-1,0,1],[4838,9E+09,9E+09,9E+09,9E+09,9E+09]],[[296.823,39.1379,95.3469],[0.138102,0.693464,0.693504,-0.138156],[-1,-1,0,1],[4838,9E+09,9E+09,9E+09,9E+09,9E+09]],[[296.852,27.3436,102.215],[0.092318,0.70103,0.701076,-0.0923436],[-1,-1,0,1],[4838,9E+09,9E+09,9E+09,9E+09,9E+09]],[[296.829,13.7895,104.903],[0.0462517,0.705607,0.705577,-0.0462699],[-1,0,-1,0],[4838,9E+09,9E+09,9E+09,9E+09,9E+09]],[[296.839,0.00979208,105.095],[2.40556E-05,-0.707095,-0.707119,-6.38552E-07],[-1,0,-1,0],[4838,9E+09,9E+09,9E+09,9E+09,9E+09]],[[75.54,-110.49,75.53],[0.104911,-0.592891,0.59209,0.535634],[-1,-2,0,1],[3747.5,9E+09,9E+09,9E+09,9E+09,9E+09]],[[75.54,-110.49,75.53],[0.104911,-0.592891,0.59209,0.535634],[-1,0,-1,0],[3747.5,9E+09,9E+09,9E+09,9E+09,9E+09]],[[75.54,-110.49,75.53],[0.104911,-0.592891,0.59209,0.535634],[-1,0,-1,0],[3747.5,9E+09,9E+09,9E+09,9E+09,9E+09]],[[75.54,-110.49,75.53],[0.104911,-0.592891,0.59209,0.535634],[-1,0,-1,0],[3747.5,9E+09,9E+09,9E+09,9E+09,9E+09]],[[75.54,-110.49,75.53],[0.104911,-0.592891,0.59209,0.535634],[-1,0,-1,0],[3747.5,9E+09,9E+09,9E+09,9E+09,9E+09]],[[75.54,-110.49,75.53],[0.104911,-0.592891,0.59209,0.535634],[-1,0,-1,0],[3747.5,9E+09,9E+09,9E+09,9E+09,9E+09]],[[75.54,-110.49,75.53],[0.104911,-0.592891,0.59209,0.535634],[-1,0,-1,0],[3747.5,9E+09,9E+09,9E+09,9E+09,9E+09]],[[75.54,-110.49,75.53],[0.104911,-0.592891,0.59209,0.535634],[-1,0,-1,0],[3747.5,9E+09,9E+09,9E+09,9E+09,9E+09]],[[75.54,-110.49,75.53],[0.104911,-0.592891,0.59209,0.535634],[-1,0,-1,0],[3747.5,9E+09,9E+09,9E+09,9E+09,9E+09]],[[75.54,-110.49,75.53],[0.104911,-0.592891,0.59209,0.535634],[-1,0,-1,0],[3747.5,9E+09,9E+09,9E+09,9E+09,9E+09]],[[75.54,-110.49,75.53],[0.104911,-0.592891,0.59209,0.535634],[-1,0,-1,0],[3747.5,9E+09,9E+09,9E+09,9E+09,9E+09]],[[75.54,-110.49,75.53],[0.104911,-0.592891,0.59209,0.535634],[-1,0,-1,0],[3747.5,9E+09,9E+09,9E+09,9E+09,9E+09]],[[75.54,-110.49,75.53],[0.104911,-0.592891,0.59209,0.535634],[-1,0,-1,0],[3747.5,9E+09,9E+09,9E+09,9E+09,9E+09]],[[75.54,-110.49,75.53],[0.104911,-0.592891,0.59209,0.535634],[-1,0,-1,0],[3747.5,9E+09,9E+09,9E+09,9E+09,9E+09]],[[75.54,-110.49,75.53],[0.104911,-0.592891,0.59209,0.535634],[-1,0,-1,0],[3747.5,9E+09,9E+09,9E+09,9E+09,9E+09]],[[75.54,-110.49,75.53],[0.104911,-0.592891,0.59209,0.535634],[-1,0,-1,0],[3747.5,9E+09,9E+09,9E+09,9E+09,9E+09]],[[75.54,-110.49,75.53],[0.104911,-0.592891,0.59209,0.535634],[-1,0,-1,0],[3747.5,9E+09,9E+09,9E+09,9E+09,9E+09]],[[75.54,-110.49,75.53],[0.104911,-0.592891,0.59209,0.535634],[-1,0,-1,0],[3747.5,9E+09,9E+09,9E+09,9E+09,9E+09]],[[75.54,-110.49,75.53],[0.104911,-0.592891,0.59209,0.535634],[-1,0,-1,0],[3747.5,9E+09,9E+09,9E+09,9E+09,9E+09]],[[75.54,-110.49,75.53],[0.104911,-0.592891,0.59209,0.535634],[-1,0,-1,0],[3747.5,9E+09,9E+09,9E+09,9E+09,9E+09]],[[75.54,-110.49,75.53],[0.104911,-0.592891,0.59209,0.535634],[-1,0,-1,0],[3747.5,9E+09,9E+09,9E+09,9E+09,9E+09]],[[75.54,-110.49,75.53],[0.104911,-0.592891,0.59209,0.535634],[-1,0,-1,0],[3747.5,9E+09,9E+09,9E+09,9E+09,9E+09]],[[75.54,-110.49,75.53],[0.104911,-0.592891,0.59209,0.535634],[-1,0,-1,0],[3747.5,9E+09,9E+09,9E+09,9E+09,9E+09]],[[75.54,-110.49,75.53],[0.104911,-0.592891,0.59209,0.535634],[-1,0,-1,0],[3747.5,9E+09,9E+09,9E+09,9E+09,9E+09]],[[75.54,-110.49,75.53],[0.104911,-0.592891,0.59209,0.535634],[-1,0,-1,0],[3747.5,9E+09,9E+09,9E+09,9E+09,9E+09]],[[75.54,-110.49,75.53],[0.104911,-0.592891,0.59209,0.535634],[-1,0,-1,0],[3747.5,9E+09,9E+09,9E+09,9E+09,9E+09]],[[75.54,-110.49,75.53],[0.104911,-0.592891,0.59209,0.535634],[-1,0,-1,0],[3747.5,9E+09,9E+09,9E+09,9E+09,9E+09]],[[75.54,-110.49,75.53],[0.104911,-0.592891,0.59209,0.535634],[-1,0,-1,0],[3747.5,9E+09,9E+09,9E+09,9E+09,9E+09]],[[75.54,-110.49,75.53],[0.104911,-0.592891,0.59209,0.535634],[-1,0,-1,0],[3747.5,9E+09,9E+09,9E+09,9E+09,9E+09]],[[75.54,-110.49,75.53],[0.104911,-0.592891,0.59209,0.535634],[-1,0,-1,0],[3747.5,9E+09,9E+09,9E+09,9E+09,9E+09]],[[75.54,-110.49,75.53],[0.104911,-0.592891,0.59209,0.535634],[-1,0,-1,0],[3747.5,9E+09,9E+09,9E+09,9E+09,9E+09]],[[75.54,-110.49,75.53],[0.104911,-0.592891,0.59209,0.535634],[-1,0,-1,0],[3747.5,9E+09,9E+09,9E+09,9E+09,9E+09]],[[75.54,-110.49,75.53],[0.104911,-0.592891,0.59209,0.535634],[-1,0,-1,0],[3747.5,9E+09,9E+09,9E+09,9E+09,9E+09]],[[75.54,-110.49,75.53],[0.104911,-0.592891,0.59209,0.535634],[-1,0,-1,0],[3747.5,9E+09,9E+09,9E+09,9E+09,9E+09]],[[75.54,-110.49,75.53],[0.104911,-0.592891,0.59209,0.535634],[-1,0,-1,0],[3747.5,9E+09,9E+09,9E+09,9E+09,9E+09]],[[75.54,-110.49,75.53],[0.104911,-0.592891,0.59209,0.535634],[-1,0,-1,0],[3747.5,9E+09,9E+09,9E+09,9E+09,9E+09]],[[75.54,-110.49,75.53],[0.104911,-0.592891,0.59209,0.535634],[-1,0,-1,0],[3747.5,9E+09,9E+09,9E+09,9E+09,9E+09]],[[75.54,-110.49,75.53],[0.104911,-0.592891,0.59209,0.535634],[-1,0,-1,0],[3747.5,9E+09,9E+09,9E+09,9E+09,9E+09]],[[75.54,-110.49,75.53],[0.104911,-0.592891,0.59209,0.535634],[-1,0,-1,0],[3747.5,9E+09,9E+09,9E+09,9E+09,9E+09]],[[75.54,-110.49,75.53],[0.104911,-0.592891,0.59209,0.535634],[-1,0,-1,0],[3747.5,9E+09,9E+09,9E+09,9E+09,9E+09]],[[75.54,-110.49,75.53],[0.104911,-0.592891,0.59209,0.535634],[-1,0,-1,0],[3747.5,9E+09,9E+09,9E+09,9E+09,9E+09]],[[75.54,-110.49,75.53],[0.104911,-0.592891,0.59209,0.535634],[-1,0,-1,0],[3747.5,9E+09,9E+09,9E+09,9E+09,9E+09]],[[75.54,-110.49,75.53],[0.104911,-0.592891,0.59209,0.535634],[-1,0,-1,0],[3747.5,9E+09,9E+09,9E+09,9E+09,9E+09]],[[75.54,-110.49,75.53],[0.104911,-0.592891,0.59209,0.535634],[-1,0,-1,0],[3747.5,9E+09,9E+09,9E+09,9E+09,9E+09]],[[75.54,-110.49,75.53],[0.104911,-0.592891,0.59209,0.535634],[-1,0,-1,0],[3747.5,9E+09,9E+09,9E+09,9E+09,9E+09]],[[75.54,-110.49,75.53],[0.104911,-0.592891,0.59209,0.535634],[-1,0,-1,0],[3747.5,9E+09,9E+09,9E+09,9E+09,9E+09]],[[75.54,-110.49,75.53],[0.104911,-0.592891,0.59209,0.535634],[-1,0,-1,0],[3747.5,9E+09,9E+09,9E+09,9E+09,9E+09]],[[75.54,-110.49,75.53],[0.104911,-0.592891,0.59209,0.535634],[-1,0,-1,0],[3747.5,9E+09,9E+09,9E+09,9E+09,9E+09]],[[75.54,-110.49,75.53],[0.104911,-0.592891,0.59209,0.535634],[-1,0,-1,0],[3747.5,9E+09,9E+09,9E+09,9E+09,9E+09]],[[75.54,-110.49,75.53],[0.104911,-0.592891,0.59209,0.535634],[-1,0,-1,0],[3747.5,9E+09,9E+09,9E+09,9E+09,9E+09]],[[75.54,-110.49,75.53],[0.104911,-0.592891,0.59209,0.535634],[-1,0,-1,0],[3747.5,9E+09,9E+09,9E+09,9E+09,9E+09]],[[75.54,-110.49,75.53],[0.104911,-0.592891,0.59209,0.535634],[-1,0,-1,0],[3747.5,9E+09,9E+09,9E+09,9E+09,9E+09]],[[75.54,-110.49,75.53],[0.104911,-0.592891,0.59209,0.535634],[-1,0,-1,0],[3747.5,9E+09,9E+09,9E+09,9E+09,9E+09]],[[75.54,-110.49,75.53],[0.104911,-0.592891,0.59209,0.535634],[-1,0,-1,0],[3747.5,9E+09,9E+09,9E+09,9E+09,9E+09]],[[75.54,-110.49,75.53],[0.104911,-0.592891,0.59209,0.535634],[-1,0,-1,0],[3747.5,9E+09,9E+09,9E+09,9E+09,9E+09]],[[75.54,-110.49,75.53],[0.104911,-0.592891,0.59209,0.535634],[-1,0,-1,0],[3747.5,9E+09,9E+09,9E+09,9E+09,9E+09]],[[75.54,-110.49,75.53],[0.104911,-0.592891,0.59209,0.535634],[-1,0,-1,0],[3747.5,9E+09,9E+09,9E+09,9E+09,9E+09]],[[75.54,-110.49,75.53],[0.104911,-0.592891,0.59209,0.535634],[-1,0,-1,0],[3747.5,9E+09,9E+09,9E+09,9E+09,9E+09]],[[75.54,-110.49,75.53],[0.104911,-0.592891,0.59209,0.535634],[-1,0,-1,0],[3747.5,9E+09,9E+09,9E+09,9E+09,9E+09]],[[75.54,-110.49,75.53],[0.104911,-0.592891,0.59209,0.535634],[-1,0,-1,0],[3747.5,9E+09,9E+09,9E+09,9E+09,9E+09]],[[75.54,-110.49,75.53],[0.104911,-0.592891,0.59209,0.535634],[-1,0,-1,0],[3747.5,9E+09,9E+09,9E+09,9E+09,9E+09]],[[75.54,-110.49,75.53],[0.104911,-0.592891,0.59209,0.535634],[-1,0,-1,0],[3747.5,9E+09,9E+09,9E+09,9E+09,9E+09]],[[75.54,-110.49,75.53],[0.104911,-0.592891,0.59209,0.535634],[-1,0,-1,0],[3747.5,9E+09,9E+09,9E+09,9E+09,9E+09]],[[75.54,-110.49,75.53],[0.104911,-0.592891,0.59209,0.535634],[-1,0,-1,0],[3747.5,9E+09,9E+09,9E+09,9E+09,9E+09]],[[75.54,-110.49,75.53],[0.104911,-0.592891,0.59209,0.535634],[-1,0,-1,0],[3747.5,9E+09,9E+09,9E+09,9E+09,9E+09]],[[75.54,-110.49,75.53],[0.104911,-0.592891,0.59209,0.535634],[-1,0,-1,0],[3747.5,9E+09,9E+09,9E+09,9E+09,9E+09]],[[75.54,-110.49,75.53],[0.104911,-0.592891,0.59209,0.535634],[-1,0,-1,0],[3747.5,9E+09,9E+09,9E+09,9E+09,9E+09]],[[75.54,-110.49,75.53],[0.104911,-0.592891,0.59209,0.535634],[-1,0,-1,0],[3747.5,9E+09,9E+09,9E+09,9E+09,9E+09]],[[75.54,-110.49,75.53],[0.104911,-0.592891,0.59209,0.535634],[-1,0,-1,0],[3747.5,9E+09,9E+09,9E+09,9E+09,9E+09]],[[75.54,-110.49,75.53],[0.104911,-0.592891,0.59209,0.535634],[-1,0,-1,0],[3747.5,9E+09,9E+09,9E+09,9E+09,9E+09]],[[75.54,-110.49,75.53],[0.104911,-0.592891,0.59209,0.535634],[-1,0,-1,0],[3747.5,9E+09,9E+09,9E+09,9E+09,9E+09]],[[75.54,-110.49,75.53],[0.104911,-0.592891,0.59209,0.535634],[-1,0,-1,0],[3747.5,9E+09,9E+09,9E+09,9E+09,9E+09]],[[75.54,-110.49,75.53],[0.104911,-0.592891,0.59209,0.535634],[-1,0,-1,0],[3747.5,9E+09,9E+09,9E+09,9E+09,9E+09]],[[75.54,-110.49,75.53],[0.104911,-0.592891,0.59209,0.535634],[-1,0,-1,0],[3747.5,9E+09,9E+09,9E+09,9E+09,9E+09]],[[75.54,-110.49,75.53],[0.104911,-0.592891,0.59209,0.535634],[-1,0,-1,0],[3747.5,9E+09,9E+09,9E+09,9E+09,9E+09]],[[75.54,-110.49,75.53],[0.104911,-0.592891,0.59209,0.535634],[-1,0,-1,0],[3747.5,9E+09,9E+09,9E+09,9E+09,9E+09]],[[75.54,-110.49,75.53],[0.104911,-0.592891,0.59209,0.535634],[-1,0,-1,0],[3747.5,9E+09,9E+09,9E+09,9E+09,9E+09]],[[75.54,-110.49,75.53],[0.104911,-0.592891,0.59209,0.535634],[-1,0,-1,0],[3747.5,9E+09,9E+09,9E+09,9E+09,9E+09]],[[75.54,-110.49,75.53],[0.104911,-0.592891,0.59209,0.535634],[-1,0,-1,0],[3747.5,9E+09,9E+09,9E+09,9E+09,9E+09]],[[75.54,-110.49,75.53],[0.104911,-0.592891,0.59209,0.535634],[-1,0,-1,0],[3747.5,9E+09,9E+09,9E+09,9E+09,9E+09]],[[75.54,-110.49,75.53],[0.104911,-0.592891,0.59209,0.535634],[-1,0,-1,0],[3747.5,9E+09,9E+09,9E+09,9E+09,9E+09]],[[75.54,-110.49,75.53],[0.104911,-0.592891,0.59209,0.535634],[-1,0,-1,0],[3747.5,9E+09,9E+09,9E+09,9E+09,9E+09]],[[75.54,-110.49,75.53],[0.104911,-0.592891,0.59209,0.535634],[-1,0,-1,0],[3747.5,9E+09,9E+09,9E+09,9E+09,9E+09]],[[75.54,-110.49,75.53],[0.104911,-0.592891,0.59209,0.535634],[-1,0,-1,0],[3747.5,9E+09,9E+09,9E+09,9E+09,9E+09]],[[75.54,-110.49,75.53],[0.104911,-0.592891,0.59209,0.535634],[-1,0,-1,0],[3747.5,9E+09,9E+09,9E+09,9E+09,9E+09]],[[75.54,-110.49,75.53],[0.104911,-0.592891,0.59209,0.535634],[-1,0,-1,0],[3747.5,9E+09,9E+09,9E+09,9E+09,9E+09]],[[75.54,-110.49,75.53],[0.104911,-0.592891,0.59209,0.535634],[-1,0,-1,0],[3747.5,9E+09,9E+09,9E+09,9E+09,9E+09]]];
    TASK PERS pos posSSHPeripherys{100}:=[[1189.26,-121.425,101.165],[1189.26,-122.75,98.2787],[1189.26,-125.534,95.4221],[1189.32,-79.2411,121.281],[1189.27,-104.291,118.451],[1189.25,-108.25,115.514],[1189.25,-111.327,112.696],[1189.26,-112.495,109.743],[1189.27,-114.688,106.925],[1189.26,-118.942,103.987],[1189.26,-121.425,101.165],[1189.26,-122.75,98.2787],[1189.26,-125.534,95.4221],[1189.26,-127.439,92.439],[1189.26,-130.079,89.5448],[1189.27,-131.245,86.7067],[1189.28,-133.292,83.8021],[1189.28,-135.789,80.9103],[1189.28,-137.388,78.0515],[1189.28,-138.406,75.2576],[1189.28,-139.427,72.3021],[1189.27,-141.483,69.4441],[1189.28,-142.219,66.5296],[1189.28,-143.389,63.6236],[1189.28,-145.296,60.7212],[1189.29,-145.888,57.7957],[1189.29,-146.897,54.8963],[1189.3,-148.648,52.0778],[1189.28,-149.405,49.1086],[1189.28,-150.723,46.2847],[1189.28,-151.444,43.3672],[1189.28,-152.915,40.4255],[1189.28,-153.646,37.465],[1189.28,-153.495,34.6376],[1189.29,-154.96,31.7538],[1189.29,-155.406,28.9001],[1189.29,-156.001,25.9568],[1189.29,-156.441,23.0264],[1189.28,-156.589,20.2191],[1189.29,-156.423,17.2819],[1189.29,-157.151,14.4496],[1189.28,-158.041,11.5136],[1189.28,-158.044,8.70987],[1189.28,-157.906,5.7459],[1189.28,-158.345,2.80928],[1189.29,-158.194,-0.0186222],[1189.29,-160.83,-2.92115],[1189.3,-158.038,-5.85137],[1189.29,-157.892,-8.68883],[1189.29,-157.747,-11.5968],[1189.27,-157.906,-14.5726],[1189.28,-157.313,-17.3681],[1189.27,-156.442,-20.3021],[1189.29,-156.568,-23.1149],[1189.29,-155.552,-26.0754],[1189.28,-155.562,-28.9223],[1189.29,-154.976,-31.8306],[1189.28,-154.092,-34.7765],[1189.28,-153.492,-37.5781],[1189.29,-152.895,-40.4902],[1189.28,-152.317,-43.4585],[1189.28,-152.477,-46.2586],[1189.27,-150.579,-49.2274],[1189.27,-149.851,-52.0675],[1189.28,-148.218,-54.9559],[1189.28,-147.643,-57.9081],[1189.28,-146.039,-60.7614],[1189.28,-145.169,-63.6491],[1189.27,-144.292,-66.6197],[1189.27,-143.254,-69.4298],[1189.28,-141.772,-72.3288],[1189.26,-139.305,-75.298],[1189.26,-139.312,-78.1109],[1189.26,-137.12,-81.0493],[1189.27,-134.327,-84.4392],[1189.27,-134.023,-86.8162],[1189.28,-131.815,-89.7404],[1189.28,-130.07,-92.561],[1189.28,-79.2253,-95.4585],[1189.27,-125.682,-98.2712],[1189.27,-123.617,-101.205],[1189.26,-79.2201,-104.06],[1189.26,-118.055,-106.977],[1189.26,-115.847,-109.906],[1189.26,-111.183,-112.759],[1189.26,-108.387,-115.688],[1189.26,-79.2458,-118.493],[1189.26,-103.564,-121.442],[1189.25,-101.095,-124.428],[1189.25,-79.2612,-127.228],[462.156,-67.387,-88.0007],[462.953,-64.1692,-88.6888],[0,0,0],[0,0,0],[0,0,0],[0,0,0],[0,0,0],[0,0,0],[0,0,0],[0,0,0]];
    TASK PERS robtarget robtSSHPeripheryCenter:=[[1189.23,-158.521,-0.436458],[0.500015,-0.500005,-0.499989,-0.499991],[-1,-1,-3,1],[4202,9E+09,9E+09,9E+09,9E+09,9E+09]];
    TASK PERS pose poseSSHPeripheryCenter:=[[-0.0150146,0.729416,0.0185326],[1,0,0,0]];

    TASK PERS jointtarget jointSSApproach:=[[0,-45,45,0,60,0],[4837,9E+09,9E+09,9E+09,9E+09,9E+09]];
    TASK PERS jointtarget jointSSDepart:=[[0,-45,45,0,60,0],[4837,9E+09,9E+09,9E+09,9E+09,9E+09]];

    VAR iodev iodevSSBLog;
    VAR iodev iodevSSHLog;

    TASK PERS num numSSHLLSInterval:=0.103616;
    TASK PERS num numSSHLLSScan:=90;
    TASK PERS pos posSSHLLSClosest:=[1189.29,-160.83,-2.92115];
    TASK PERS num numSSHLLSClosestLaseValue:=-31.6126;
    TASK PERS num numSSHLLSClosestIndex:=47;
    VAR intnum intSSHLinerLaserScan;

    TASK PERS num numSSBLLSInterval:=0.104032;
    TASK PERS num numSSBLLSScan:=90;
    TASK PERS pos posSSBLLSClosest:=[388.11,-58.601,218.152];
    TASK PERS num numSSBLLSClosestLaseValue:=31.3959;
    TASK PERS num numSSBLLSClosestIndex:=39;
    VAR intnum intSSBLinerLaserScan;


    CONST string strSPBLogFileName:="ScanPlatoonBranch1.csv";
    CONST string strSPHLogFileName:="ScanPlatoonHeader1.csv";

    !For platoon branch SmarTac
    TASK PERS num numSPBPointsTotal:=13;
    !Scan platoon branch range
    TASK PERS num numSPBAngleFrom:=220;
    TASK PERS num numSPBAngleTo:=320;

    !For platoon header SmarTac
    TASK PERS num numSPHPointsTotal:=13;
    !Scan platoon header range
    TASK PERS num numSPHAngleFrom:=180;
    TASK PERS num numSPHAngleTo:=120;

    !Scan platoon branch points
    TASK PERS robtarget robtSPBLaserSmarTacs{20}:=[[[3740.81,-24.4902,293.7],[0.241845,-0.664463,-0.241845,-0.664463],[0,0,-2,1],[1447,9E+09,9E+09,9E+09,9E+09,9E+09]],[[3744.67,-28.4617,293.7],[0.289484,-0.645135,-0.289484,-0.645135],[0,0,-2,1],[1447,9E+09,9E+09,9E+09,9E+09,9E+09]],[[3749.06,-31.8321,293.7],[0.335593,-0.622396,-0.335593,-0.622396],[0,0,-1,1],[1447,9E+09,9E+09,9E+09,9E+09,9E+09]],[[3753.9,-34.5303,293.7],[0.379928,-0.596368,-0.379928,-0.596368],[0,0,-1,1],[1447,9E+09,9E+09,9E+09,9E+09,9E+09]],[[3759.07,-36.4994,293.7],[0.422255,-0.567187,-0.422255,-0.567187],[0,0,-1,1],[1447,9E+09,9E+09,9E+09,9E+09,9E+09]],[[3764.48,-37.6977,293.7],[0.462349,-0.535007,-0.462349,-0.535007],[0,0,-1,1],[1447,9E+09,9E+09,9E+09,9E+09,9E+09]],[[3770,-38.1,293.7],[0.5,-0.5,-0.5,-0.5],[0,-1,1,1],[1447,9E+09,9E+09,9E+09,9E+09,9E+09]],[[3775.52,-37.6977,293.7],[0.535007,-0.462349,-0.535008,-0.462349],[-1,-1,1,1],[1447,9E+09,9E+09,9E+09,9E+09,9E+09]],[[3780.93,-36.4994,293.7],[0.567187,-0.422255,-0.567187,-0.422255],[-1,-1,1,1],[1447,9E+09,9E+09,9E+09,9E+09,9E+09]],[[3786.1,-34.5303,293.7],[0.596368,-0.379928,-0.596368,-0.379928],[-1,-1,1,1],[1447,9E+09,9E+09,9E+09,9E+09,9E+09]],[[3790.94,-31.8321,293.7],[0.622396,-0.335593,-0.622396,-0.335593],[-1,-1,1,1],[1447,9E+09,9E+09,9E+09,9E+09,9E+09]],[[3795.33,-28.4617,293.7],[0.645135,-0.289484,-0.645135,-0.289484],[-1,-1,1,1],[1447,9E+09,9E+09,9E+09,9E+09,9E+09]],[[3799.19,-24.4902,293.7],[0.664463,-0.241845,-0.664463,-0.241845],[-1,-1,1,1],[1447,9E+09,9E+09,9E+09,9E+09,9E+09]],[[652.53,-493.33,1047.99],[0.459259,-0.544323,-0.447932,-0.54051],[-1,-1,1,1],[4837,9E+09,9E+09,9E+09,9E+09,9E+09]],[[652.53,-493.33,1047.99],[0.459259,-0.544323,-0.447932,-0.54051],[-1,0,-2,1],[4837,9E+09,9E+09,9E+09,9E+09,9E+09]],[[652.53,-493.33,1047.99],[0.459259,-0.544323,-0.447932,-0.54051],[-1,0,-2,1],[4837,9E+09,9E+09,9E+09,9E+09,9E+09]],[[652.53,-493.33,1047.99],[0.459259,-0.544323,-0.447932,-0.54051],[-1,0,-2,1],[4837,9E+09,9E+09,9E+09,9E+09,9E+09]],[[652.53,-493.33,1047.99],[0.459259,-0.544323,-0.447932,-0.54051],[-1,0,-2,1],[4837,9E+09,9E+09,9E+09,9E+09,9E+09]],[[652.53,-493.33,1047.99],[0.459259,-0.544323,-0.447932,-0.54051],[-1,0,-2,1],[4837,9E+09,9E+09,9E+09,9E+09,9E+09]],[[652.53,-493.33,1047.99],[0.459259,-0.544323,-0.447932,-0.54051],[-1,0,-2,1],[4837,9E+09,9E+09,9E+09,9E+09,9E+09]]];
    TASK PERS robtarget robtSPBWireSmarTacs{20}:=[[[428.493,28.575,188.15],[0.683013,0.183013,-0.683013,0.183013],[0,1,-3,1],[4838,9E+09,9E+09,9E+09,9E+09,9E+09]],[[422.779,36.7353,188.15],[0.664463,0.241845,-0.664463,0.241845],[0,1,-3,1],[4838,9E+09,9E+09,9E+09,9E+09,9E+09]],[[415.735,43.7794,188.15],[0.640856,0.298836,-0.640856,0.298836],[0,1,-3,1],[4838,9E+09,9E+09,9E+09,9E+09,9E+09]],[[407.575,49.4934,188.15],[0.612372,0.353553,-0.612372,0.353553],[0,0,-3,1],[4838,9E+09,9E+09,9E+09,9E+09,9E+09]],[[398.546,53.7034,188.15],[0.579228,0.40558,-0.579228,0.40558],[0,0,-3,1],[4838,9E+09,9E+09,9E+09,9E+09,9E+09]],[[388.924,56.2818,188.15],[0.541675,0.454519,-0.541675,0.454519],[0,0,-3,1],[4838,9E+09,9E+09,9E+09,9E+09,9E+09]],[[379,57.15,188.15],[0.5,0.5,-0.5,0.5],[0,0,-3,1],[4838,9E+09,9E+09,9E+09,9E+09,9E+09]],[[369.076,56.2818,188.15],[0.454519,0.541675,-0.454519,0.541675],[-1,-1,-2,1],[4838,9E+09,9E+09,9E+09,9E+09,9E+09]],[[359.454,53.7034,188.15],[0.40558,0.579228,-0.40558,0.579228],[-1,-1,-2,1],[4838,9E+09,9E+09,9E+09,9E+09,9E+09]],[[350.425,49.4934,188.15],[0.353553,0.612372,-0.353553,0.612372],[-1,-1,-2,1],[4838,9E+09,9E+09,9E+09,9E+09,9E+09]],[[342.265,43.7794,188.15],[0.298836,0.640856,-0.298836,0.640856],[-1,-2,-2,1],[4838,9E+09,9E+09,9E+09,9E+09,9E+09]],[[335.221,36.7353,188.15],[0.241845,0.664463,-0.241845,0.664463],[-1,-2,-2,1],[4838,9E+09,9E+09,9E+09,9E+09,9E+09]],[[329.507,28.575,188.15],[0.183013,0.683013,-0.183013,0.683013],[-1,-2,-2,1],[4838,9E+09,9E+09,9E+09,9E+09,9E+09]],[[652.53,-493.33,1047.99],[0.459259,-0.544323,-0.447932,-0.54051],[-1,-1,-2,1],[4837,9E+09,9E+09,9E+09,9E+09,9E+09]],[[652.53,-493.33,1047.99],[0.459259,-0.544323,-0.447932,-0.54051],[-1,0,-2,1],[4837,9E+09,9E+09,9E+09,9E+09,9E+09]],[[652.53,-493.33,1047.99],[0.459259,-0.544323,-0.447932,-0.54051],[-1,0,-2,1],[4837,9E+09,9E+09,9E+09,9E+09,9E+09]],[[652.53,-493.33,1047.99],[0.459259,-0.544323,-0.447932,-0.54051],[-1,0,-2,1],[4837,9E+09,9E+09,9E+09,9E+09,9E+09]],[[652.53,-493.33,1047.99],[0.459259,-0.544323,-0.447932,-0.54051],[-1,0,-2,1],[4837,9E+09,9E+09,9E+09,9E+09,9E+09]],[[652.53,-493.33,1047.99],[0.459259,-0.544323,-0.447932,-0.54051],[-1,0,-2,1],[4837,9E+09,9E+09,9E+09,9E+09,9E+09]],[[652.53,-493.33,1047.99],[0.459259,-0.544323,-0.447932,-0.54051],[-1,0,-2,1],[4837,9E+09,9E+09,9E+09,9E+09,9E+09]]];
    TASK PERS robtarget robtSPBLinerFrom:=[[3274.49,-38.1,268.15],[3.09086E-08,3.09086E-08,-0.707107,-0.707107],[0,0,1,1],[1967,9E+09,9E+09,9E+09,9E+09,9E+09]];
    TASK PERS robtarget robtSPBLinerTo:=[[3225.51,-38.1,268.15],[3.09086E-08,3.09086E-08,-0.707107,-0.707107],[0,0,1,1],[1967,9E+09,9E+09,9E+09,9E+09,9E+09]];

    !Scan platoon branch results, shared for all the four scan methods
    TASK PERS pose poseSPBs{20}:=[[[0.671631,0.571692,-0.0139771],[1,0,0,0]],[[1.48047,1.70094,0.0154724],[1,0,0,0]],[[0.750488,1.14403,0.00900269],[1,0,0,0]],[[0.697266,1.46957,0.0152283],[1,0,0,0]],[[0.488037,1.70678,0.0148315],[1,0,0,0]],[[0.0710449,0.546875,0.00549316],[1,0,0,0]],[[-0.00415039,1.56931,-0.0259399],[1,0,0,0]],[[-0.0671387,0.53194,0.0257874],[1,0,0,0]],[[-0.151611,0.435173,0.00985718],[1,0,0,0]],[[-0.519531,1.0752,-0.000640869],[1,0,0,0]],[[0.685059,-1.00649,0.0101013],[1,0,0,0]],[[0.254883,-0.304142,-0.0348206],[1,0,0,0]],[[0.294922,-0.246531,0.0117188],[1,0,0,0]],[[0,0,0],[1,0,0,0]],[[0,0,0],[1,0,0,0]],[[0,0,0],[1,0,0,0]],[[0,0,0],[1,0,0,0]],[[0,0,0],[1,0,0,0]],[[0,0,0],[1,0,0,0]],[[0,0,0],[1,0,0,0]]];
    TASK PERS num numSPBLaserValues{100}:=[-0.547806,-0.108337,0.331123,-0.547806,-0.547806,-0.547806,-0.108337,-0.547806,-0.547806,-0.254829,-0.254829,0.331123,-0.547806,0,0,0,0,0,0,0,0,0,0,0,0,0,0,0,0,0,0,0,0,0,0,0,0,0,0,0,0,0,0,0,0,0,0,0,0,0,0,0,0,0,0,0,0,0,0,0,0,0,0,0,0,0,0,0,0,0,0,0,0,0,0,0,0,0,0,0,0,0,0,0,0,0,0,0,0,0,0,0,0,0,0,0,0,0,0,0];
    TASK PERS robtarget robtSPBPeripherys{100}:=[[[2246.07,-24.2706,268.136],[0.640854,-0.640863,0.298826,-0.29884],[0,0,-2,1],[2942,9E+09,9E+09,9E+09,9E+09,9E+09]],[[2251.08,-26.8416,268.165],[0.660882,-0.660874,0.25148,-0.251472],[0,0,-2,1],[2942,9E+09,9E+09,9E+09,9E+09,9E+09]],[[2255,-30.4114,268.159],[0.677413,-0.677392,0.2028,-0.202792],[0,0,-1,1],[2942,9E+09,9E+09,9E+09,9E+09,9E+09]],[[2259.36,-33.5572,268.165],[0.690351,-0.690338,0.153031,-0.153072],[0,0,-1,1],[2942,9E+09,9E+09,9E+09,9E+09,9E+09]],[[2264.4,-35.3174,268.165],[0.699649,-0.699636,0.102462,-0.102483],[0,0,-1,1],[2942,9E+09,9E+09,9E+09,9E+09,9E+09]],[[2269.47,-37.6929,268.155],[0.705239,-0.705236,0.0513691,-0.0513853],[0,0,-1,1],[2942,9E+09,9E+09,9E+09,9E+09,9E+09]],[[2275,-36.639,268.124],[7.62567E-06,-7.48469E-06,-0.707124,-0.70709],[0,-1,1,1],[2942,9E+09,9E+09,9E+09,9E+09,9E+09]],[[2280.53,-37.7078,268.176],[0.0513794,0.0513753,-0.705232,-0.705244],[-1,-1,1,1],[2942,9E+09,9E+09,9E+09,9E+09,9E+09]],[[2285.93,-36.589,268.16],[0.102496,0.102493,-0.699636,-0.699642],[-1,-1,1,1],[2941.99,9E+09,9E+09,9E+09,9E+09,9E+09]],[[2290.69,-33.6861,268.149],[0.153047,0.153055,-0.690345,-0.690343],[-1,-1,1,1],[2942,9E+09,9E+09,9E+09,9E+09,9E+09]],[[2296.76,-33.0515,268.16],[0.202775,0.202813,-0.677401,-0.677405],[-1,-1,1,1],[2942,9E+09,9E+09,9E+09,9E+09,9E+09]],[[2300.36,-28.5184,268.115],[0.251489,0.251475,-0.660897,-0.660854],[-1,-1,1,1],[2942,9E+09,9E+09,9E+09,9E+09,9E+09]],[[2304.9,-25.0889,268.162],[0.298833,0.298843,-0.640854,-0.640857],[-1,-1,1,1],[2942,9E+09,9E+09,9E+09,9E+09,9E+09]],[[75.54,-110.49,75.53],[0.104911,-0.592891,0.59209,0.535634],[-1,-2,0,1],[3747.5,9E+09,9E+09,9E+09,9E+09,9E+09]],[[75.54,-110.49,75.53],[0.104911,-0.592891,0.59209,0.535634],[-1,0,-1,0],[3747.5,9E+09,9E+09,9E+09,9E+09,9E+09]],[[75.54,-110.49,75.53],[0.104911,-0.592891,0.59209,0.535634],[-1,0,-1,0],[3747.5,9E+09,9E+09,9E+09,9E+09,9E+09]],[[75.54,-110.49,75.53],[0.104911,-0.592891,0.59209,0.535634],[-1,0,-1,0],[3747.5,9E+09,9E+09,9E+09,9E+09,9E+09]],[[75.54,-110.49,75.53],[0.104911,-0.592891,0.59209,0.535634],[-1,0,-1,0],[3747.5,9E+09,9E+09,9E+09,9E+09,9E+09]],[[75.54,-110.49,75.53],[0.104911,-0.592891,0.59209,0.535634],[-1,0,-1,0],[3747.5,9E+09,9E+09,9E+09,9E+09,9E+09]],[[75.54,-110.49,75.53],[0.104911,-0.592891,0.59209,0.535634],[-1,0,-1,0],[3747.5,9E+09,9E+09,9E+09,9E+09,9E+09]],[[75.54,-110.49,75.53],[0.104911,-0.592891,0.59209,0.535634],[-1,0,-1,0],[3747.5,9E+09,9E+09,9E+09,9E+09,9E+09]],[[75.54,-110.49,75.53],[0.104911,-0.592891,0.59209,0.535634],[-1,0,-1,0],[3747.5,9E+09,9E+09,9E+09,9E+09,9E+09]],[[75.54,-110.49,75.53],[0.104911,-0.592891,0.59209,0.535634],[-1,0,-1,0],[3747.5,9E+09,9E+09,9E+09,9E+09,9E+09]],[[75.54,-110.49,75.53],[0.104911,-0.592891,0.59209,0.535634],[-1,0,-1,0],[3747.5,9E+09,9E+09,9E+09,9E+09,9E+09]],[[75.54,-110.49,75.53],[0.104911,-0.592891,0.59209,0.535634],[-1,0,-1,0],[3747.5,9E+09,9E+09,9E+09,9E+09,9E+09]],[[75.54,-110.49,75.53],[0.104911,-0.592891,0.59209,0.535634],[-1,0,-1,0],[3747.5,9E+09,9E+09,9E+09,9E+09,9E+09]],[[75.54,-110.49,75.53],[0.104911,-0.592891,0.59209,0.535634],[-1,0,-1,0],[3747.5,9E+09,9E+09,9E+09,9E+09,9E+09]],[[75.54,-110.49,75.53],[0.104911,-0.592891,0.59209,0.535634],[-1,0,-1,0],[3747.5,9E+09,9E+09,9E+09,9E+09,9E+09]],[[75.54,-110.49,75.53],[0.104911,-0.592891,0.59209,0.535634],[-1,0,-1,0],[3747.5,9E+09,9E+09,9E+09,9E+09,9E+09]],[[75.54,-110.49,75.53],[0.104911,-0.592891,0.59209,0.535634],[-1,0,-1,0],[3747.5,9E+09,9E+09,9E+09,9E+09,9E+09]],[[75.54,-110.49,75.53],[0.104911,-0.592891,0.59209,0.535634],[-1,0,-1,0],[3747.5,9E+09,9E+09,9E+09,9E+09,9E+09]],[[75.54,-110.49,75.53],[0.104911,-0.592891,0.59209,0.535634],[-1,0,-1,0],[3747.5,9E+09,9E+09,9E+09,9E+09,9E+09]],[[75.54,-110.49,75.53],[0.104911,-0.592891,0.59209,0.535634],[-1,0,-1,0],[3747.5,9E+09,9E+09,9E+09,9E+09,9E+09]],[[75.54,-110.49,75.53],[0.104911,-0.592891,0.59209,0.535634],[-1,0,-1,0],[3747.5,9E+09,9E+09,9E+09,9E+09,9E+09]],[[75.54,-110.49,75.53],[0.104911,-0.592891,0.59209,0.535634],[-1,0,-1,0],[3747.5,9E+09,9E+09,9E+09,9E+09,9E+09]],[[75.54,-110.49,75.53],[0.104911,-0.592891,0.59209,0.535634],[-1,0,-1,0],[3747.5,9E+09,9E+09,9E+09,9E+09,9E+09]],[[75.54,-110.49,75.53],[0.104911,-0.592891,0.59209,0.535634],[-1,0,-1,0],[3747.5,9E+09,9E+09,9E+09,9E+09,9E+09]],[[75.54,-110.49,75.53],[0.104911,-0.592891,0.59209,0.535634],[-1,0,-1,0],[3747.5,9E+09,9E+09,9E+09,9E+09,9E+09]],[[75.54,-110.49,75.53],[0.104911,-0.592891,0.59209,0.535634],[-1,0,-1,0],[3747.5,9E+09,9E+09,9E+09,9E+09,9E+09]],[[75.54,-110.49,75.53],[0.104911,-0.592891,0.59209,0.535634],[-1,0,-1,0],[3747.5,9E+09,9E+09,9E+09,9E+09,9E+09]],[[75.54,-110.49,75.53],[0.104911,-0.592891,0.59209,0.535634],[-1,0,-1,0],[3747.5,9E+09,9E+09,9E+09,9E+09,9E+09]],[[75.54,-110.49,75.53],[0.104911,-0.592891,0.59209,0.535634],[-1,0,-1,0],[3747.5,9E+09,9E+09,9E+09,9E+09,9E+09]],[[75.54,-110.49,75.53],[0.104911,-0.592891,0.59209,0.535634],[-1,0,-1,0],[3747.5,9E+09,9E+09,9E+09,9E+09,9E+09]],[[75.54,-110.49,75.53],[0.104911,-0.592891,0.59209,0.535634],[-1,0,-1,0],[3747.5,9E+09,9E+09,9E+09,9E+09,9E+09]],[[75.54,-110.49,75.53],[0.104911,-0.592891,0.59209,0.535634],[-1,0,-1,0],[3747.5,9E+09,9E+09,9E+09,9E+09,9E+09]],[[75.54,-110.49,75.53],[0.104911,-0.592891,0.59209,0.535634],[-1,0,-1,0],[3747.5,9E+09,9E+09,9E+09,9E+09,9E+09]],[[75.54,-110.49,75.53],[0.104911,-0.592891,0.59209,0.535634],[-1,0,-1,0],[3747.5,9E+09,9E+09,9E+09,9E+09,9E+09]],[[75.54,-110.49,75.53],[0.104911,-0.592891,0.59209,0.535634],[-1,0,-1,0],[3747.5,9E+09,9E+09,9E+09,9E+09,9E+09]],[[75.54,-110.49,75.53],[0.104911,-0.592891,0.59209,0.535634],[-1,0,-1,0],[3747.5,9E+09,9E+09,9E+09,9E+09,9E+09]],[[75.54,-110.49,75.53],[0.104911,-0.592891,0.59209,0.535634],[-1,0,-1,0],[3747.5,9E+09,9E+09,9E+09,9E+09,9E+09]],[[75.54,-110.49,75.53],[0.104911,-0.592891,0.59209,0.535634],[-1,0,-1,0],[3747.5,9E+09,9E+09,9E+09,9E+09,9E+09]],[[75.54,-110.49,75.53],[0.104911,-0.592891,0.59209,0.535634],[-1,0,-1,0],[3747.5,9E+09,9E+09,9E+09,9E+09,9E+09]],[[75.54,-110.49,75.53],[0.104911,-0.592891,0.59209,0.535634],[-1,0,-1,0],[3747.5,9E+09,9E+09,9E+09,9E+09,9E+09]],[[75.54,-110.49,75.53],[0.104911,-0.592891,0.59209,0.535634],[-1,0,-1,0],[3747.5,9E+09,9E+09,9E+09,9E+09,9E+09]],[[75.54,-110.49,75.53],[0.104911,-0.592891,0.59209,0.535634],[-1,0,-1,0],[3747.5,9E+09,9E+09,9E+09,9E+09,9E+09]],[[75.54,-110.49,75.53],[0.104911,-0.592891,0.59209,0.535634],[-1,0,-1,0],[3747.5,9E+09,9E+09,9E+09,9E+09,9E+09]],[[75.54,-110.49,75.53],[0.104911,-0.592891,0.59209,0.535634],[-1,0,-1,0],[3747.5,9E+09,9E+09,9E+09,9E+09,9E+09]],[[75.54,-110.49,75.53],[0.104911,-0.592891,0.59209,0.535634],[-1,0,-1,0],[3747.5,9E+09,9E+09,9E+09,9E+09,9E+09]],[[75.54,-110.49,75.53],[0.104911,-0.592891,0.59209,0.535634],[-1,0,-1,0],[3747.5,9E+09,9E+09,9E+09,9E+09,9E+09]],[[75.54,-110.49,75.53],[0.104911,-0.592891,0.59209,0.535634],[-1,0,-1,0],[3747.5,9E+09,9E+09,9E+09,9E+09,9E+09]],[[75.54,-110.49,75.53],[0.104911,-0.592891,0.59209,0.535634],[-1,0,-1,0],[3747.5,9E+09,9E+09,9E+09,9E+09,9E+09]],[[75.54,-110.49,75.53],[0.104911,-0.592891,0.59209,0.535634],[-1,0,-1,0],[3747.5,9E+09,9E+09,9E+09,9E+09,9E+09]],[[75.54,-110.49,75.53],[0.104911,-0.592891,0.59209,0.535634],[-1,0,-1,0],[3747.5,9E+09,9E+09,9E+09,9E+09,9E+09]],[[75.54,-110.49,75.53],[0.104911,-0.592891,0.59209,0.535634],[-1,0,-1,0],[3747.5,9E+09,9E+09,9E+09,9E+09,9E+09]],[[75.54,-110.49,75.53],[0.104911,-0.592891,0.59209,0.535634],[-1,0,-1,0],[3747.5,9E+09,9E+09,9E+09,9E+09,9E+09]],[[75.54,-110.49,75.53],[0.104911,-0.592891,0.59209,0.535634],[-1,0,-1,0],[3747.5,9E+09,9E+09,9E+09,9E+09,9E+09]],[[75.54,-110.49,75.53],[0.104911,-0.592891,0.59209,0.535634],[-1,0,-1,0],[3747.5,9E+09,9E+09,9E+09,9E+09,9E+09]],[[75.54,-110.49,75.53],[0.104911,-0.592891,0.59209,0.535634],[-1,0,-1,0],[3747.5,9E+09,9E+09,9E+09,9E+09,9E+09]],[[75.54,-110.49,75.53],[0.104911,-0.592891,0.59209,0.535634],[-1,0,-1,0],[3747.5,9E+09,9E+09,9E+09,9E+09,9E+09]],[[75.54,-110.49,75.53],[0.104911,-0.592891,0.59209,0.535634],[-1,0,-1,0],[3747.5,9E+09,9E+09,9E+09,9E+09,9E+09]],[[75.54,-110.49,75.53],[0.104911,-0.592891,0.59209,0.535634],[-1,0,-1,0],[3747.5,9E+09,9E+09,9E+09,9E+09,9E+09]],[[75.54,-110.49,75.53],[0.104911,-0.592891,0.59209,0.535634],[-1,0,-1,0],[3747.5,9E+09,9E+09,9E+09,9E+09,9E+09]],[[75.54,-110.49,75.53],[0.104911,-0.592891,0.59209,0.535634],[-1,0,-1,0],[3747.5,9E+09,9E+09,9E+09,9E+09,9E+09]],[[75.54,-110.49,75.53],[0.104911,-0.592891,0.59209,0.535634],[-1,0,-1,0],[3747.5,9E+09,9E+09,9E+09,9E+09,9E+09]],[[75.54,-110.49,75.53],[0.104911,-0.592891,0.59209,0.535634],[-1,0,-1,0],[3747.5,9E+09,9E+09,9E+09,9E+09,9E+09]],[[75.54,-110.49,75.53],[0.104911,-0.592891,0.59209,0.535634],[-1,0,-1,0],[3747.5,9E+09,9E+09,9E+09,9E+09,9E+09]],[[75.54,-110.49,75.53],[0.104911,-0.592891,0.59209,0.535634],[-1,0,-1,0],[3747.5,9E+09,9E+09,9E+09,9E+09,9E+09]],[[75.54,-110.49,75.53],[0.104911,-0.592891,0.59209,0.535634],[-1,0,-1,0],[3747.5,9E+09,9E+09,9E+09,9E+09,9E+09]],[[75.54,-110.49,75.53],[0.104911,-0.592891,0.59209,0.535634],[-1,0,-1,0],[3747.5,9E+09,9E+09,9E+09,9E+09,9E+09]],[[75.54,-110.49,75.53],[0.104911,-0.592891,0.59209,0.535634],[-1,0,-1,0],[3747.5,9E+09,9E+09,9E+09,9E+09,9E+09]],[[75.54,-110.49,75.53],[0.104911,-0.592891,0.59209,0.535634],[-1,0,-1,0],[3747.5,9E+09,9E+09,9E+09,9E+09,9E+09]],[[75.54,-110.49,75.53],[0.104911,-0.592891,0.59209,0.535634],[-1,0,-1,0],[3747.5,9E+09,9E+09,9E+09,9E+09,9E+09]],[[75.54,-110.49,75.53],[0.104911,-0.592891,0.59209,0.535634],[-1,0,-1,0],[3747.5,9E+09,9E+09,9E+09,9E+09,9E+09]],[[75.54,-110.49,75.53],[0.104911,-0.592891,0.59209,0.535634],[-1,0,-1,0],[3747.5,9E+09,9E+09,9E+09,9E+09,9E+09]],[[75.54,-110.49,75.53],[0.104911,-0.592891,0.59209,0.535634],[-1,0,-1,0],[3747.5,9E+09,9E+09,9E+09,9E+09,9E+09]],[[75.54,-110.49,75.53],[0.104911,-0.592891,0.59209,0.535634],[-1,0,-1,0],[3747.5,9E+09,9E+09,9E+09,9E+09,9E+09]],[[75.54,-110.49,75.53],[0.104911,-0.592891,0.59209,0.535634],[-1,0,-1,0],[3747.5,9E+09,9E+09,9E+09,9E+09,9E+09]],[[75.54,-110.49,75.53],[0.104911,-0.592891,0.59209,0.535634],[-1,0,-1,0],[3747.5,9E+09,9E+09,9E+09,9E+09,9E+09]],[[75.54,-110.49,75.53],[0.104911,-0.592891,0.59209,0.535634],[-1,0,-1,0],[3747.5,9E+09,9E+09,9E+09,9E+09,9E+09]],[[75.54,-110.49,75.53],[0.104911,-0.592891,0.59209,0.535634],[-1,0,-1,0],[3747.5,9E+09,9E+09,9E+09,9E+09,9E+09]],[[75.54,-110.49,75.53],[0.104911,-0.592891,0.59209,0.535634],[-1,0,-1,0],[3747.5,9E+09,9E+09,9E+09,9E+09,9E+09]],[[75.54,-110.49,75.53],[0.104911,-0.592891,0.59209,0.535634],[-1,0,-1,0],[3747.5,9E+09,9E+09,9E+09,9E+09,9E+09]],[[75.54,-110.49,75.53],[0.104911,-0.592891,0.59209,0.535634],[-1,0,-1,0],[3747.5,9E+09,9E+09,9E+09,9E+09,9E+09]],[[75.54,-110.49,75.53],[0.104911,-0.592891,0.59209,0.535634],[-1,0,-1,0],[3747.5,9E+09,9E+09,9E+09,9E+09,9E+09]],[[75.54,-110.49,75.53],[0.104911,-0.592891,0.59209,0.535634],[-1,0,-1,0],[3747.5,9E+09,9E+09,9E+09,9E+09,9E+09]],[[75.54,-110.49,75.53],[0.104911,-0.592891,0.59209,0.535634],[-1,0,-1,0],[3747.5,9E+09,9E+09,9E+09,9E+09,9E+09]],[[75.54,-110.49,75.53],[0.104911,-0.592891,0.59209,0.535634],[-1,0,-1,0],[3747.5,9E+09,9E+09,9E+09,9E+09,9E+09]],[[75.54,-110.49,75.53],[0.104911,-0.592891,0.59209,0.535634],[-1,0,-1,0],[3747.5,9E+09,9E+09,9E+09,9E+09,9E+09]],[[75.54,-110.49,75.53],[0.104911,-0.592891,0.59209,0.535634],[-1,0,-1,0],[3747.5,9E+09,9E+09,9E+09,9E+09,9E+09]],[[75.54,-110.49,75.53],[0.104911,-0.592891,0.59209,0.535634],[-1,0,-1,0],[3747.5,9E+09,9E+09,9E+09,9E+09,9E+09]]];
    TASK PERS pos posSPBPeripherys{100}:=[[3268.46,-36.3091,268.076],[3267.87,-37.0478,268.074],[3267.25,-37.1903,268.089],[3266.67,-37.0417,268.112],[3266.03,-37.1838,268.127],[3265.44,-37.6193,268.138],[3264.84,-38.206,268.141],[3264.22,-38.2057,268.144],[3263.65,-37.6219,268.141],[3263.03,-38.9399,268.139],[3262.01,-38.9386,268.142],[3261.81,-38.9376,268.143],[3261.18,-39.0818,268.143],[3260.61,-38.9363,268.145],[3259.99,-39.376,268.145],[3259.39,-39.0825,268.146],[3258.82,-39.5233,268.147],[3258.18,-39.0847,268.147],[3257.62,-39.2314,268.148],[3257,-39.9633,268.151],[3256.38,-39.5243,268.151],[3255.79,-39.8176,268.152],[3255.15,-40.1118,268.15],[3254.58,-39.8188,268.152],[3253.98,-39.5269,268.149],[3253.34,-39.8193,268.154],[3252.74,-39.382,268.151],[3252.13,-39.9691,268.152],[3251.55,-39.8243,268.151],[3250.97,-39.0946,268.152],[3250.33,-39.3896,268.151],[3249.75,-39.8329,268.151],[3249.14,-39.5422,268.151],[3248.54,-39.5452,268.152],[3247.95,-39.4013,268.154],[3247.31,-39.111,268.156],[3246.73,-39.4058,268.159],[3246.12,-39.1108,268.164],[3245.55,-39.1076,268.172],[3244.97,-38.9594,268.176],[3244.32,-38.6645,268.184],[3243.75,-38.3673,268.192],[3243.14,-38.6563,268.202],[3242.52,-38.6523,268.208],[3241.94,-38.0608,268.218],[3241.31,-37.6158,268.227],[3240.73,-37.4682,268.229],[3240.13,-37.1718,268.237],[3239.52,-36.7304,268.237],[3238.94,-36.5819,268.238],[3238.31,-36.2901,268.228],[3237.74,-36.4356,268.221],[3237.14,-35.5574,268.21],[3236.37,-35.5593,268.2],[3235.93,-35.4124,268.194],[3235.29,-34.8255,268.191],[3234.7,-34.6842,268.18],[3234.14,-34.3936,268.178],[3233.51,-34.3927,268.174],[3232.93,-33.8102,268.167],[3232.31,11.9044,268.165],[3231.73,11.9039,268.156],[3231.14,11.9024,268.15],[3230.5,11.903,268.152],[3229.93,11.9041,268.156],[3229.32,11.902,268.156],[3228.72,11.902,268.159],[3228.15,11.9028,268.157],[3227.51,11.903,268.156],[3226.93,11.9064,268.158],[3226.33,11.904,268.152],[3225.71,11.9034,268.15],[3231.14,11.9024,268.15],[3230.5,11.903,268.152],[3229.93,11.9041,268.156],[3229.32,11.902,268.156],[3228.72,11.902,268.159],[3228.15,11.9028,268.157],[3227.51,11.903,268.156],[3226.93,11.9064,268.158],[3226.33,11.904,268.152],[3225.71,11.9034,268.15],[3272.52,-38.645,268.154],[3271.94,-38.9374,268.154],[3271.33,-38.2026,268.151],[3270.7,-37.6166,268.151],[3270.12,-38.0561,268.151],[3269.51,-37.3223,268.153],[3268.92,-37.1766,268.153],[3268.33,-37.4725,268.148],[332.054,-39.994,188.152],[0,0,0],[0,0,0],[0,0,0],[0,0,0],[0,0,0],[0,0,0],[0,0,0],[0,0,0],[0,0,0]];
    TASK PERS robtarget robtSPBPeripheryCenter:=[[3253.43,-39.5811,268.149],[2.07492E-05,1.93905E-05,-0.707106,-0.707108],[0,-1,1,1],[1967,9E+09,9E+09,9E+09,9E+09,9E+09]];
    TASK PERS pose poseSPBPeripheryCenter:=[[-0.0349121,-1.48106,-0.00112915],[1,0,0,0]];

    !Scan platoon header points
    TASK PERS robtarget robtSPHLaserSmarTacs{20}:=[[[2703.1,-133.7,-1.16884E-05],[0.5,-0.5,0.5,0.5],[0,-1,0,1],[2602,9E+09,9E+09,9E+09,9E+09,9E+09]],[[2703.1,-133.191,11.6527],[0.477714,-0.521334,0.521334,0.477714],[0,-1,0,1],[2602,9E+09,9E+09,9E+09,9E+09,9E+09]],[[2703.1,-131.669,23.2168],[0.454519,-0.541675,0.541675,0.454519],[0,-1,0,1],[2602,9E+09,9E+09,9E+09,9E+09,9E+09]],[[2703.1,-129.144,34.6041],[0.430459,-0.560986,0.560986,0.430459],[0,-1,0,1],[2602,9E+09,9E+09,9E+09,9E+09,9E+09]],[[2703.1,-125.637,45.7281],[0.40558,-0.579228,0.579228,0.40558],[0,-1,0,1],[2602,9E+09,9E+09,9E+09,9E+09,9E+09]],[[2703.1,-121.173,56.5041],[0.379928,-0.596368,0.596368,0.379928],[0,-1,0,1],[2602,9E+09,9E+09,9E+09,9E+09,9E+09]],[[2703.1,-115.788,66.85],[0.353553,-0.612372,0.612372,0.353553],[0,-1,0,1],[2602,9E+09,9E+09,9E+09,9E+09,9E+09]],[[2703.1,-109.521,76.6872],[0.326506,-0.627211,0.627211,0.326506],[0,-1,0,1],[2602,9E+09,9E+09,9E+09,9E+09,9E+09]],[[2703.1,-102.42,85.9407],[0.298836,-0.640856,0.640856,0.298836],[0,-1,0,1],[2602,9E+09,9E+09,9E+09,9E+09,9E+09]],[[2703.1,-94.5402,94.5402],[0.270598,-0.653282,0.653281,0.270598],[0,-1,0,1],[2602,9E+09,9E+09,9E+09,9E+09,9E+09]],[[2703.1,-85.9407,102.42],[0.241845,-0.664463,0.664463,0.241845],[0,-1,0,1],[2602,9E+09,9E+09,9E+09,9E+09,9E+09]],[[2703.1,-76.6872,109.521],[0.212631,-0.67438,0.67438,0.212631],[0,-1,0,1],[2602,9E+09,9E+09,9E+09,9E+09,9E+09]],[[2703.1,-66.85,115.788],[0.183013,-0.683013,0.683013,0.183013],[0,0,-1,0],[2602,9E+09,9E+09,9E+09,9E+09,9E+09]],[[652.53,-493.33,1047.99],[0.459259,-0.544323,-0.447932,-0.54051],[0,0,-1,0],[4837,9E+09,9E+09,9E+09,9E+09,9E+09]],[[652.53,-493.33,1047.99],[0.459259,-0.544323,-0.447932,-0.54051],[-1,0,-2,1],[4837,9E+09,9E+09,9E+09,9E+09,9E+09]],[[652.53,-493.33,1047.99],[0.459259,-0.544323,-0.447932,-0.54051],[-1,0,-2,1],[4837,9E+09,9E+09,9E+09,9E+09,9E+09]],[[652.53,-493.33,1047.99],[0.459259,-0.544323,-0.447932,-0.54051],[-1,0,-2,1],[4837,9E+09,9E+09,9E+09,9E+09,9E+09]],[[652.53,-493.33,1047.99],[0.459259,-0.544323,-0.447932,-0.54051],[-1,0,-2,1],[4837,9E+09,9E+09,9E+09,9E+09,9E+09]],[[652.53,-493.33,1047.99],[0.459259,-0.544323,-0.447932,-0.54051],[-1,0,-2,1],[4837,9E+09,9E+09,9E+09,9E+09,9E+09]],[[652.53,-493.33,1047.99],[0.459259,-0.544323,-0.447932,-0.54051],[-1,0,-2,1],[4837,9E+09,9E+09,9E+09,9E+09,9E+09]]];
    TASK PERS robtarget robtSPHWireSmarTacs{20}:=[[[296.85,108.15,0],[0.5,0.5,-0.5,0.5],[-1,-1,2,1],[4838,9E+09,9E+09,9E+09,9E+09,9E+09]],[[296.85,107.225,14.1164],[0.466228,0.531631,-0.531631,0.466228],[-1,-1,2,1],[4838,9E+09,9E+09,9E+09,9E+09,9E+09]],[[296.85,104.465,27.9913],[0.430459,0.560986,-0.560986,0.430459],[-1,-1,2,1],[4838,9E+09,9E+09,9E+09,9E+09,9E+09]],[[296.85,99.9176,41.3872],[0.392847,0.587938,-0.587938,0.392848],[-1,0,1,0],[4838,9E+09,9E+09,9E+09,9E+09,9E+09]],[[296.85,93.6606,54.075],[0.353553,0.612372,-0.612372,0.353553],[-1,0,1,0],[4838,9E+09,9E+09,9E+09,9E+09,9E+09]],[[296.85,85.8012,65.8375],[0.312745,0.634185,-0.634185,0.312745],[-1,0,1,0],[4838,9E+09,9E+09,9E+09,9E+09,9E+09]],[[296.85,76.4736,76.4736],[0.270598,0.653282,0.653281,-0.270598],[-1,-1,0,1],[4838,9E+09,9E+09,9E+09,9E+09,9E+09]],[[296.85,65.8375,85.8012],[0.227292,0.669581,0.669581,-0.227292],[-1,-1,0,1],[4838,9E+09,9E+09,9E+09,9E+09,9E+09]],[[296.85,54.075,93.6607],[0.183013,0.683013,0.683013,-0.183013],[-1,-1,0,1],[4838,9E+09,9E+09,9E+09,9E+09,9E+09]],[[296.85,41.3872,99.9176],[0.13795,0.69352,0.69352,-0.13795],[-1,-1,0,1],[4838,9E+09,9E+09,9E+09,9E+09,9E+09]],[[296.85,27.9913,104.465],[0.092296,0.701057,0.701057,-0.092296],[-1,-1,0,1],[4838,9E+09,9E+09,9E+09,9E+09,9E+09]],[[296.85,14.1164,107.225],[0.046247,0.705593,0.705593,-0.046247],[-1,0,-1,0],[4838,9E+09,9E+09,9E+09,9E+09,9E+09]],[[296.85,-4.72739E-06,108.15],[3.09086E-08,-0.707107,-0.707107,-3.09086E-08],[-1,0,-1,0],[4838,9E+09,9E+09,9E+09,9E+09,9E+09]],[[652.53,-493.33,1047.99],[0.459259,-0.544323,-0.447932,-0.54051],[-1,0,-1,0],[4837,9E+09,9E+09,9E+09,9E+09,9E+09]],[[652.53,-493.33,1047.99],[0.459259,-0.544323,-0.447932,-0.54051],[-1,0,-2,1],[4837,9E+09,9E+09,9E+09,9E+09,9E+09]],[[652.53,-493.33,1047.99],[0.459259,-0.544323,-0.447932,-0.54051],[-1,0,-2,1],[4837,9E+09,9E+09,9E+09,9E+09,9E+09]],[[652.53,-493.33,1047.99],[0.459259,-0.544323,-0.447932,-0.54051],[-1,0,-2,1],[4837,9E+09,9E+09,9E+09,9E+09,9E+09]],[[652.53,-493.33,1047.99],[0.459259,-0.544323,-0.447932,-0.54051],[-1,0,-2,1],[4837,9E+09,9E+09,9E+09,9E+09,9E+09]],[[652.53,-493.33,1047.99],[0.459259,-0.544323,-0.447932,-0.54051],[-1,0,-2,1],[4837,9E+09,9E+09,9E+09,9E+09,9E+09]],[[652.53,-493.33,1047.99],[0.459259,-0.544323,-0.447932,-0.54051],[-1,0,-2,1],[4837,9E+09,9E+09,9E+09,9E+09,9E+09]]];
    TASK PERS robtarget robtSPHLinerFrom:=[[3338.1,-108.15,88.5913],[0.5,-0.5,0.5,0.5],[-1,-1,-1,1],[1967,9E+09,9E+09,9E+09,9E+09,9E+09]];
    TASK PERS robtarget robtSPHLinerTo:=[[3338.1,-108.15,-88.5913],[0.5,-0.5,0.5,0.5],[-1,-1,-1,1],[1967,9E+09,9E+09,9E+09,9E+09,9E+09]];

    !Scan platoon header results, shared for all the four scan methods
    TASK PERS pose poseSPHs{20}:=[[[0.00537109,-0.220146,-0.0317405],[1,0,0,0]],[[0.0112305,-1.31258,0.1263],[1,0,0,0]],[[0.00146484,-1.43652,0.300823],[1,0,0,0]],[[-0.00732422,-2.24283,0.695314],[1,0,0,0]],[[0.00146484,-2.38943,1.00131],[1,0,0,0]],[[-0.00146484,-2.80038,1.44713],[1,0,0,0]],[[0.00146484,-2.44102,1.54834],[1,0,0,0]],[[0.0356445,-3.43182,2.62237],[1,0,0,0]],[[0.00390625,-3.3073,3.0287],[1,0,0,0]],[[-0.000488281,-3.40851,4.05803],[1,0,0,0]],[[0.00195313,-2.71912,3.87146],[1,0,0,0]],[[0.0708008,-2.59956,4.64789],[1,0,0,0]],[[0.000976563,-2.44021,5.51877],[1,0,0,0]],[[0,0,0],[1,0,0,0]],[[0,0,0],[1,0,0,0]],[[0,0,0],[1,0,0,0]],[[0,0,0],[1,0,0,0]],[[0,0,0],[1,0,0,0]],[[0,0,0],[1,0,0,0]],[[0,0,0],[1,0,0,0]]];
    TASK PERS num numSPHLaserValues{100}:=[0,0,0,0,0,0,0,0,0,0,0,0,0,0,0,0,0,0,0,0,0,0,0,0,0,0,0,0,0,0,0,0,0,0,0,0,0,0,0,0,0,0,0,0,0,0,0,0,0,0,0,0,0,0,0,0,0,0,0,0,0,0,0,0,0,0,0,0,0,0,0,0,0,0,0,0,0,0,0,0,0,0,0,0,0,0,0,0,0,0,0,0,0,0,0,0,0,0,0,0];
    TASK PERS robtarget robtSPHPeripherys{100}:=[[[4121.11,-108.37,-0.03175],[0.499998,-0.500013,0.500003,0.499985],[0,-1,0,1],[1159,9E+09,9E+09,9E+09,9E+09,9E+09]],[[4121.11,-108.965,10.492],[0.475434,-0.523407,0.52342,0.475435],[0,-1,0,1],[1159,9E+09,9E+09,9E+09,9E+09,9E+09]],[[4121.1,-107.6,20.9368],[0.449773,-0.545616,0.545625,0.449779],[0,-1,0,1],[1159,9E+09,9E+09,9E+09,9E+09,9E+09]],[[4121.09,-105.939,31.4116],[0.423084,-0.566564,0.566566,0.423093],[0,-1,0,1],[1159,9E+09,9E+09,9E+09,9E+09,9E+09]],[[4121.1,-102.664,41.515],[0.395424,-0.586215,0.586205,0.395417],[0,-1,0,1],[1159,9E+09,9E+09,9E+09,9E+09,9E+09]],[[4121.1,-98.7306,51.3853],[0.36682,-0.604514,0.604522,0.366822],[0,-1,0,1],[1159,9E+09,9E+09,9E+09,9E+09,9E+09]],[[4121.1,-93.1432,60.4511],[0.337397,-0.621416,0.621424,0.337398],[0,-1,0,1],[1159,9E+09,9E+09,9E+09,9E+09,9E+09]],[[4121.14,-88.0709,69.9473],[0.307213,-0.636965,0.636856,0.307099],[0,-1,0,1],[1159,9E+09,9E+09,9E+09,9E+09,9E+09]],[[4121.1,-81.1039,78.156],[0.276239,-0.65094,0.650903,0.276215],[0,-1,0,1],[1159,9E+09,9E+09,9E+09,9E+09,9E+09]],[[4121.1,-73.6463,86.2959],[0.244757,-0.663404,0.663389,0.244755],[0,-1,0,1],[1159,9E+09,9E+09,9E+09,9E+09,9E+09]],[[4121.1,-64.7514,92.4628],[0.212627,-0.674381,0.674382,0.212624],[0,-1,0,1],[1159,9E+09,9E+09,9E+09,9E+09,9E+09]],[[4121.17,-55.8552,98.7769],[0.180077,-0.683791,0.683812,0.18001],[0,-1,0,1],[1159,9E+09,9E+09,9E+09,9E+09,9E+09]],[[4121.1,-46.4288,104.319],[0.147019,-0.691657,0.691651,0.147019],[0,0,-1,0],[1159,9E+09,9E+09,9E+09,9E+09,9E+09]],[[75.54,-110.49,75.53],[0.104911,-0.592891,0.59209,0.535634],[-1,-2,0,1],[3747.5,9E+09,9E+09,9E+09,9E+09,9E+09]],[[75.54,-110.49,75.53],[0.104911,-0.592891,0.59209,0.535634],[-1,0,-1,0],[3747.5,9E+09,9E+09,9E+09,9E+09,9E+09]],[[75.54,-110.49,75.53],[0.104911,-0.592891,0.59209,0.535634],[-1,0,-1,0],[3747.5,9E+09,9E+09,9E+09,9E+09,9E+09]],[[75.54,-110.49,75.53],[0.104911,-0.592891,0.59209,0.535634],[-1,0,-1,0],[3747.5,9E+09,9E+09,9E+09,9E+09,9E+09]],[[75.54,-110.49,75.53],[0.104911,-0.592891,0.59209,0.535634],[-1,0,-1,0],[3747.5,9E+09,9E+09,9E+09,9E+09,9E+09]],[[75.54,-110.49,75.53],[0.104911,-0.592891,0.59209,0.535634],[-1,0,-1,0],[3747.5,9E+09,9E+09,9E+09,9E+09,9E+09]],[[75.54,-110.49,75.53],[0.104911,-0.592891,0.59209,0.535634],[-1,0,-1,0],[3747.5,9E+09,9E+09,9E+09,9E+09,9E+09]],[[75.54,-110.49,75.53],[0.104911,-0.592891,0.59209,0.535634],[-1,0,-1,0],[3747.5,9E+09,9E+09,9E+09,9E+09,9E+09]],[[75.54,-110.49,75.53],[0.104911,-0.592891,0.59209,0.535634],[-1,0,-1,0],[3747.5,9E+09,9E+09,9E+09,9E+09,9E+09]],[[75.54,-110.49,75.53],[0.104911,-0.592891,0.59209,0.535634],[-1,0,-1,0],[3747.5,9E+09,9E+09,9E+09,9E+09,9E+09]],[[75.54,-110.49,75.53],[0.104911,-0.592891,0.59209,0.535634],[-1,0,-1,0],[3747.5,9E+09,9E+09,9E+09,9E+09,9E+09]],[[75.54,-110.49,75.53],[0.104911,-0.592891,0.59209,0.535634],[-1,0,-1,0],[3747.5,9E+09,9E+09,9E+09,9E+09,9E+09]],[[75.54,-110.49,75.53],[0.104911,-0.592891,0.59209,0.535634],[-1,0,-1,0],[3747.5,9E+09,9E+09,9E+09,9E+09,9E+09]],[[75.54,-110.49,75.53],[0.104911,-0.592891,0.59209,0.535634],[-1,0,-1,0],[3747.5,9E+09,9E+09,9E+09,9E+09,9E+09]],[[75.54,-110.49,75.53],[0.104911,-0.592891,0.59209,0.535634],[-1,0,-1,0],[3747.5,9E+09,9E+09,9E+09,9E+09,9E+09]],[[75.54,-110.49,75.53],[0.104911,-0.592891,0.59209,0.535634],[-1,0,-1,0],[3747.5,9E+09,9E+09,9E+09,9E+09,9E+09]],[[75.54,-110.49,75.53],[0.104911,-0.592891,0.59209,0.535634],[-1,0,-1,0],[3747.5,9E+09,9E+09,9E+09,9E+09,9E+09]],[[75.54,-110.49,75.53],[0.104911,-0.592891,0.59209,0.535634],[-1,0,-1,0],[3747.5,9E+09,9E+09,9E+09,9E+09,9E+09]],[[75.54,-110.49,75.53],[0.104911,-0.592891,0.59209,0.535634],[-1,0,-1,0],[3747.5,9E+09,9E+09,9E+09,9E+09,9E+09]],[[75.54,-110.49,75.53],[0.104911,-0.592891,0.59209,0.535634],[-1,0,-1,0],[3747.5,9E+09,9E+09,9E+09,9E+09,9E+09]],[[75.54,-110.49,75.53],[0.104911,-0.592891,0.59209,0.535634],[-1,0,-1,0],[3747.5,9E+09,9E+09,9E+09,9E+09,9E+09]],[[75.54,-110.49,75.53],[0.104911,-0.592891,0.59209,0.535634],[-1,0,-1,0],[3747.5,9E+09,9E+09,9E+09,9E+09,9E+09]],[[75.54,-110.49,75.53],[0.104911,-0.592891,0.59209,0.535634],[-1,0,-1,0],[3747.5,9E+09,9E+09,9E+09,9E+09,9E+09]],[[75.54,-110.49,75.53],[0.104911,-0.592891,0.59209,0.535634],[-1,0,-1,0],[3747.5,9E+09,9E+09,9E+09,9E+09,9E+09]],[[75.54,-110.49,75.53],[0.104911,-0.592891,0.59209,0.535634],[-1,0,-1,0],[3747.5,9E+09,9E+09,9E+09,9E+09,9E+09]],[[75.54,-110.49,75.53],[0.104911,-0.592891,0.59209,0.535634],[-1,0,-1,0],[3747.5,9E+09,9E+09,9E+09,9E+09,9E+09]],[[75.54,-110.49,75.53],[0.104911,-0.592891,0.59209,0.535634],[-1,0,-1,0],[3747.5,9E+09,9E+09,9E+09,9E+09,9E+09]],[[75.54,-110.49,75.53],[0.104911,-0.592891,0.59209,0.535634],[-1,0,-1,0],[3747.5,9E+09,9E+09,9E+09,9E+09,9E+09]],[[75.54,-110.49,75.53],[0.104911,-0.592891,0.59209,0.535634],[-1,0,-1,0],[3747.5,9E+09,9E+09,9E+09,9E+09,9E+09]],[[75.54,-110.49,75.53],[0.104911,-0.592891,0.59209,0.535634],[-1,0,-1,0],[3747.5,9E+09,9E+09,9E+09,9E+09,9E+09]],[[75.54,-110.49,75.53],[0.104911,-0.592891,0.59209,0.535634],[-1,0,-1,0],[3747.5,9E+09,9E+09,9E+09,9E+09,9E+09]],[[75.54,-110.49,75.53],[0.104911,-0.592891,0.59209,0.535634],[-1,0,-1,0],[3747.5,9E+09,9E+09,9E+09,9E+09,9E+09]],[[75.54,-110.49,75.53],[0.104911,-0.592891,0.59209,0.535634],[-1,0,-1,0],[3747.5,9E+09,9E+09,9E+09,9E+09,9E+09]],[[75.54,-110.49,75.53],[0.104911,-0.592891,0.59209,0.535634],[-1,0,-1,0],[3747.5,9E+09,9E+09,9E+09,9E+09,9E+09]],[[75.54,-110.49,75.53],[0.104911,-0.592891,0.59209,0.535634],[-1,0,-1,0],[3747.5,9E+09,9E+09,9E+09,9E+09,9E+09]],[[75.54,-110.49,75.53],[0.104911,-0.592891,0.59209,0.535634],[-1,0,-1,0],[3747.5,9E+09,9E+09,9E+09,9E+09,9E+09]],[[75.54,-110.49,75.53],[0.104911,-0.592891,0.59209,0.535634],[-1,0,-1,0],[3747.5,9E+09,9E+09,9E+09,9E+09,9E+09]],[[75.54,-110.49,75.53],[0.104911,-0.592891,0.59209,0.535634],[-1,0,-1,0],[3747.5,9E+09,9E+09,9E+09,9E+09,9E+09]],[[75.54,-110.49,75.53],[0.104911,-0.592891,0.59209,0.535634],[-1,0,-1,0],[3747.5,9E+09,9E+09,9E+09,9E+09,9E+09]],[[75.54,-110.49,75.53],[0.104911,-0.592891,0.59209,0.535634],[-1,0,-1,0],[3747.5,9E+09,9E+09,9E+09,9E+09,9E+09]],[[75.54,-110.49,75.53],[0.104911,-0.592891,0.59209,0.535634],[-1,0,-1,0],[3747.5,9E+09,9E+09,9E+09,9E+09,9E+09]],[[75.54,-110.49,75.53],[0.104911,-0.592891,0.59209,0.535634],[-1,0,-1,0],[3747.5,9E+09,9E+09,9E+09,9E+09,9E+09]],[[75.54,-110.49,75.53],[0.104911,-0.592891,0.59209,0.535634],[-1,0,-1,0],[3747.5,9E+09,9E+09,9E+09,9E+09,9E+09]],[[75.54,-110.49,75.53],[0.104911,-0.592891,0.59209,0.535634],[-1,0,-1,0],[3747.5,9E+09,9E+09,9E+09,9E+09,9E+09]],[[75.54,-110.49,75.53],[0.104911,-0.592891,0.59209,0.535634],[-1,0,-1,0],[3747.5,9E+09,9E+09,9E+09,9E+09,9E+09]],[[75.54,-110.49,75.53],[0.104911,-0.592891,0.59209,0.535634],[-1,0,-1,0],[3747.5,9E+09,9E+09,9E+09,9E+09,9E+09]],[[75.54,-110.49,75.53],[0.104911,-0.592891,0.59209,0.535634],[-1,0,-1,0],[3747.5,9E+09,9E+09,9E+09,9E+09,9E+09]],[[75.54,-110.49,75.53],[0.104911,-0.592891,0.59209,0.535634],[-1,0,-1,0],[3747.5,9E+09,9E+09,9E+09,9E+09,9E+09]],[[75.54,-110.49,75.53],[0.104911,-0.592891,0.59209,0.535634],[-1,0,-1,0],[3747.5,9E+09,9E+09,9E+09,9E+09,9E+09]],[[75.54,-110.49,75.53],[0.104911,-0.592891,0.59209,0.535634],[-1,0,-1,0],[3747.5,9E+09,9E+09,9E+09,9E+09,9E+09]],[[75.54,-110.49,75.53],[0.104911,-0.592891,0.59209,0.535634],[-1,0,-1,0],[3747.5,9E+09,9E+09,9E+09,9E+09,9E+09]],[[75.54,-110.49,75.53],[0.104911,-0.592891,0.59209,0.535634],[-1,0,-1,0],[3747.5,9E+09,9E+09,9E+09,9E+09,9E+09]],[[75.54,-110.49,75.53],[0.104911,-0.592891,0.59209,0.535634],[-1,0,-1,0],[3747.5,9E+09,9E+09,9E+09,9E+09,9E+09]],[[75.54,-110.49,75.53],[0.104911,-0.592891,0.59209,0.535634],[-1,0,-1,0],[3747.5,9E+09,9E+09,9E+09,9E+09,9E+09]],[[75.54,-110.49,75.53],[0.104911,-0.592891,0.59209,0.535634],[-1,0,-1,0],[3747.5,9E+09,9E+09,9E+09,9E+09,9E+09]],[[75.54,-110.49,75.53],[0.104911,-0.592891,0.59209,0.535634],[-1,0,-1,0],[3747.5,9E+09,9E+09,9E+09,9E+09,9E+09]],[[75.54,-110.49,75.53],[0.104911,-0.592891,0.59209,0.535634],[-1,0,-1,0],[3747.5,9E+09,9E+09,9E+09,9E+09,9E+09]],[[75.54,-110.49,75.53],[0.104911,-0.592891,0.59209,0.535634],[-1,0,-1,0],[3747.5,9E+09,9E+09,9E+09,9E+09,9E+09]],[[75.54,-110.49,75.53],[0.104911,-0.592891,0.59209,0.535634],[-1,0,-1,0],[3747.5,9E+09,9E+09,9E+09,9E+09,9E+09]],[[75.54,-110.49,75.53],[0.104911,-0.592891,0.59209,0.535634],[-1,0,-1,0],[3747.5,9E+09,9E+09,9E+09,9E+09,9E+09]],[[75.54,-110.49,75.53],[0.104911,-0.592891,0.59209,0.535634],[-1,0,-1,0],[3747.5,9E+09,9E+09,9E+09,9E+09,9E+09]],[[75.54,-110.49,75.53],[0.104911,-0.592891,0.59209,0.535634],[-1,0,-1,0],[3747.5,9E+09,9E+09,9E+09,9E+09,9E+09]],[[75.54,-110.49,75.53],[0.104911,-0.592891,0.59209,0.535634],[-1,0,-1,0],[3747.5,9E+09,9E+09,9E+09,9E+09,9E+09]],[[75.54,-110.49,75.53],[0.104911,-0.592891,0.59209,0.535634],[-1,0,-1,0],[3747.5,9E+09,9E+09,9E+09,9E+09,9E+09]],[[75.54,-110.49,75.53],[0.104911,-0.592891,0.59209,0.535634],[-1,0,-1,0],[3747.5,9E+09,9E+09,9E+09,9E+09,9E+09]],[[75.54,-110.49,75.53],[0.104911,-0.592891,0.59209,0.535634],[-1,0,-1,0],[3747.5,9E+09,9E+09,9E+09,9E+09,9E+09]],[[75.54,-110.49,75.53],[0.104911,-0.592891,0.59209,0.535634],[-1,0,-1,0],[3747.5,9E+09,9E+09,9E+09,9E+09,9E+09]],[[75.54,-110.49,75.53],[0.104911,-0.592891,0.59209,0.535634],[-1,0,-1,0],[3747.5,9E+09,9E+09,9E+09,9E+09,9E+09]],[[75.54,-110.49,75.53],[0.104911,-0.592891,0.59209,0.535634],[-1,0,-1,0],[3747.5,9E+09,9E+09,9E+09,9E+09,9E+09]],[[75.54,-110.49,75.53],[0.104911,-0.592891,0.59209,0.535634],[-1,0,-1,0],[3747.5,9E+09,9E+09,9E+09,9E+09,9E+09]],[[75.54,-110.49,75.53],[0.104911,-0.592891,0.59209,0.535634],[-1,0,-1,0],[3747.5,9E+09,9E+09,9E+09,9E+09,9E+09]],[[75.54,-110.49,75.53],[0.104911,-0.592891,0.59209,0.535634],[-1,0,-1,0],[3747.5,9E+09,9E+09,9E+09,9E+09,9E+09]],[[75.54,-110.49,75.53],[0.104911,-0.592891,0.59209,0.535634],[-1,0,-1,0],[3747.5,9E+09,9E+09,9E+09,9E+09,9E+09]],[[75.54,-110.49,75.53],[0.104911,-0.592891,0.59209,0.535634],[-1,0,-1,0],[3747.5,9E+09,9E+09,9E+09,9E+09,9E+09]],[[75.54,-110.49,75.53],[0.104911,-0.592891,0.59209,0.535634],[-1,0,-1,0],[3747.5,9E+09,9E+09,9E+09,9E+09,9E+09]],[[75.54,-110.49,75.53],[0.104911,-0.592891,0.59209,0.535634],[-1,0,-1,0],[3747.5,9E+09,9E+09,9E+09,9E+09,9E+09]],[[75.54,-110.49,75.53],[0.104911,-0.592891,0.59209,0.535634],[-1,0,-1,0],[3747.5,9E+09,9E+09,9E+09,9E+09,9E+09]],[[75.54,-110.49,75.53],[0.104911,-0.592891,0.59209,0.535634],[-1,0,-1,0],[3747.5,9E+09,9E+09,9E+09,9E+09,9E+09]],[[75.54,-110.49,75.53],[0.104911,-0.592891,0.59209,0.535634],[-1,0,-1,0],[3747.5,9E+09,9E+09,9E+09,9E+09,9E+09]],[[75.54,-110.49,75.53],[0.104911,-0.592891,0.59209,0.535634],[-1,0,-1,0],[3747.5,9E+09,9E+09,9E+09,9E+09,9E+09]],[[75.54,-110.49,75.53],[0.104911,-0.592891,0.59209,0.535634],[-1,0,-1,0],[3747.5,9E+09,9E+09,9E+09,9E+09,9E+09]],[[75.54,-110.49,75.53],[0.104911,-0.592891,0.59209,0.535634],[-1,0,-1,0],[3747.5,9E+09,9E+09,9E+09,9E+09,9E+09]],[[75.54,-110.49,75.53],[0.104911,-0.592891,0.59209,0.535634],[-1,0,-1,0],[3747.5,9E+09,9E+09,9E+09,9E+09,9E+09]],[[75.54,-110.49,75.53],[0.104911,-0.592891,0.59209,0.535634],[-1,0,-1,0],[3747.5,9E+09,9E+09,9E+09,9E+09,9E+09]],[[75.54,-110.49,75.53],[0.104911,-0.592891,0.59209,0.535634],[-1,0,-1,0],[3747.5,9E+09,9E+09,9E+09,9E+09,9E+09]],[[75.54,-110.49,75.53],[0.104911,-0.592891,0.59209,0.535634],[-1,0,-1,0],[3747.5,9E+09,9E+09,9E+09,9E+09,9E+09]],[[75.54,-110.49,75.53],[0.104911,-0.592891,0.59209,0.535634],[-1,0,-1,0],[3747.5,9E+09,9E+09,9E+09,9E+09,9E+09]]];
    TASK PERS pos posSPHPeripherys{100}:=[[3338.1,-89.4958,68.7346],[3338.1,-90.2477,66.7113],[3338.1,-91.5362,64.8237],[3338.13,-76.0596,82.3092],[3338.13,-78.2342,80.4364],[3338.14,-79.8331,78.4674],[3338.14,-82.3208,76.5489],[3338.14,-83.9229,74.5731],[3338.13,-85.4071,72.6145],[3338.12,-87.0217,70.6036],[3338.1,-89.4958,68.7346],[3338.1,-90.2477,66.7113],[3338.1,-91.5362,64.8237],[3338.11,-92.7152,62.8023],[3338.11,-93.8904,60.8065],[3338.11,-95.6652,58.8825],[3338.11,-96.4016,56.8922],[3338.11,-98.1637,54.9745],[3338.1,-98.8722,53.0299],[3338.1,-99.4689,51.0697],[3338.1,-100.64,49.1076],[3338.1,-101.801,47.1308],[3338.1,-102.115,45.1998],[3338.1,-103.12,43.2107],[3338.11,-104.302,41.2029],[3338.11,-104.577,39.3116],[3338.11,-105.313,37.3073],[3338.11,-105.624,35.3667],[3338.11,-106.499,33.398],[3338.11,-107.383,31.4848],[3338.11,-107.376,29.4792],[3338.11,-108.104,27.4996],[3338.11,-109.129,25.5662],[3338.11,-109.281,23.5948],[3338.11,-109.58,21.6529],[3338.1,-110.026,19.6789],[3338.1,-110.15,17.7003],[3338.1,-110.166,15.7565],[3338.1,-111.024,13.7964],[3338.1,-110.741,11.8762],[3338.1,-110.889,9.87916],[3338.11,-110.743,7.89928],[3338.11,-111.499,5.95103],[3338.12,-111.753,4.00749],[3338.11,-111.052,2.05588],[3338.12,-112.062,0.0704858],[3338.12,-110.752,-1.83921],[3338.11,-110.015,-3.84116],[3338.12,-110.739,-5.81567],[3338.11,-110.163,-7.75527],[3338.11,-110.016,-9.74766],[3338.11,-109.28,-11.6373],[3338.11,-109.879,-13.6622],[3338.1,-108.403,-15.6257],[3338.1,-109.137,-17.54],[3338.1,-108.984,-19.5339],[3338.1,-108.69,-21.4414],[3338.1,-107.821,-23.4529],[3338.1,-107.216,-25.3309],[3338.11,-106.658,-27.3771],[3338.11,-105.464,-29.2614],[3338.11,-105.916,-31.2683],[3338.11,-105.047,-33.2061],[3338.12,-104.312,-35.1556],[3338.12,-103.133,-37.1827],[3338.12,-102.252,-39.0897],[3338.11,-102.097,-41.0757],[3338.11,-101.233,-43.0087],[3338.11,-99.3048,-44.9448],[3338.1,-99.0456,-46.9129],[3338.1,-97.8435,-48.8687],[3338.1,-96.538,-50.8727],[3338.1,-96.0932,-52.7653],[3338.1,-94.4789,-54.7574],[3338.1,-92.8631,-56.7187],[3338.1,-91.6888,-58.7228],[3338.1,-90.5177,-60.7716],[3338.1,-89.1996,-62.6643],[3338.11,-87.2957,-64.5905],[3338.11,-86.4289,-66.5333],[3338.1,-84.2252,-68.5143],[3338.1,-82.4797,-70.5366],[3338.1,-80.4085,-72.4356],[3338.09,-78.2328,-74.4399],[3338.09,-76.1556,-76.3247],[3338.09,-73.826,-78.2983],[3338.09,-72.0616,-80.2087],[3338.09,-69.4141,-82.1566],[3338.09,-67.3837,-84.1425],[3338.09,-65.0298,-86.0202],[3338.09,-61.3674,-87.9685],[1951.09,-85.064,-66.8857],[1951.12,-83.8068,-68.6542],[1951.12,-82.0627,-70.3608],[1951.11,-81.1411,-72.0366],[1951.09,-80.0304,-73.6536],[1951.09,-77.8934,-75.4358],[1951.1,-76.9367,-77.0844],[1951.11,-74.3561,-78.851],[1951.1,-73.1018,-80.5767]];
    TASK PERS robtarget robtSPHPeripheryCenter:=[[3338.09,-112.042,2.9765],[0.499978,-0.500008,0.500017,0.499997],[-1,-1,-1,1],[1967,9E+09,9E+09,9E+09,9E+09,9E+09]];
    TASK PERS pose poseSPHPeripheryCenter:=[[-0.00610352,-3.89165,-0.0112262],[1,0,0,0]];

    TASK PERS jointtarget jointSPApproach:=[[26.9156,31.391,54.477,45.4772,-61.87,-47.4425],[4837,9E+09,9E+09,9E+09,9E+09,9E+09]];
    TASK PERS jointtarget jointSPDepart:=[[2.44949,35.5941,61.0669,-0.616594,-55.163,0.115862],[4837,9E+09,9E+09,9E+09,9E+09,9E+09]];

    VAR iodev iodevSPBLog;
    VAR iodev iodevSPHLog;

    TASK PERS num numSPHLLSInterval:=0.103616;
    TASK PERS num numSPHLLSScan:=91;
    TASK PERS pos posSPHLLSClosest:=[3338.12,-112.062,0.0704858];
    TASK PERS num numSPHLLSClosestLaseValue:=-3.91705;
    TASK PERS num numSPHLLSClosestIndex:=46;
    VAR intnum intSPHLinerLaserScan;

    TASK PERS num numSPBLLSInterval:=0.1;
    TASK PERS num numSPBLLSScan:=82;
    TASK PERS pos posSPBLLSClosest:=[3255.15,-40.1118,268.15];
    TASK PERS num numSPBLLSClosestLaseValue:=-2.0127;
    TASK PERS num numSPBLLSClosestIndex:=33;
    VAR intnum intSPBLinerLaserScan;

    VAR pos center;
    VAR num radius;
    VAR pos normal;
    VAR num rms;
    VAR num maxErr;
    VAR num indexWorst;

    !For Test
    TASK PERS robtarget robtBranchCenter:=[[0,0,326.91],[1.53791E-05,0.686389,-0.727235,1.35954E-05],[-1,-1,0,0],[4837,9E+09,9E+09,9E+09,9E+09,9E+09]];
    TASK PERS robtarget robtHeaderCenter:=[[205.08,0,0],[0.648894,0.280942,-0.648906,-0.280942],[-1,0,-1,0],[4437,9E+09,9E+09,9E+09,9E+09,9E+09]];
    TASK PERS jointtarget jointBranchCenter:=[[-0.025836,21.2813,6.3797,-4.49832,26.046,7.77022],[4837,9E+09,9E+09,9E+09,9E+09,9E+09]];
    TASK PERS jointtarget jointHeaderCenter:=[[-17.3683,60.1898,-4.76592,84.4819,64.3211,-13.7158],[4437,9E+09,9E+09,9E+09,9E+09,9E+09]];
    TASK PERS robtarget robtSTN1Aligned:=[[955,-189.25,159.25],[0.489649,-0.489714,-0.510184,-0.510036],[-1,0,1,1],[4262,9E+09,9E+09,9E+09,9E+09,9E+09]];
    TASK PERS jointtarget jointSTN1Aligned:=[[-0.192923,11.1632,56.797,2.35161,-31.4728,177.014],[4202,9E+09,9E+09,9E+09,9E+09,9E+09]];

    TASK PERS robtarget robtPBCenter:=[[0,0,310],[5.16726E-05,0.708054,-0.706158,4.57025E-05],[-1,0,-1,0],[1447,9E+09,9E+09,9E+09,9E+09,9E+09]];
    TASK PERS robtarget robtPBBottom:=[[48.1,-38.1,108.15],[0.707107,-0.707107,0,0],[-1,-1,-1,1],[1337,9E+09,9E+09,9E+09,9E+09,9E+09]];
    TASK PERS robtarget robtPHCenter:=[[144.04,0,0],[0.673965,0.213937,-0.673967,-0.213939],[-1,-2,1,1],[759,9E+09,9E+09,9E+09,9E+09,9E+09]];
    TASK PERS jointtarget jointPBCenter:=[[-0.937588,28.6239,5.31149,1.86058,19.6624,-1.55408],[1447,9E+09,9E+09,9E+09,9E+09,9E+09]];
    TASK PERS jointtarget jointPBBottom:=[[-23.336,55.1725,39.7324,-59.9721,-92.8257,-92.6057],[1967,9E+09,9E+09,9E+09,9E+09,9E+09]];
    TASK PERS jointtarget jointPHCenter:=[[23.5615,77.3976,-15.0591,99.1075,-66.2014,-158.956],[2271,9E+09,9E+09,9E+09,9E+09,9E+09]];
    TASK PERS jointtarget jointPHCenter2:=[[-14.9327,76.9872,-15.1818,-97.9935,-60.7786,172.234],[759,9E+09,9E+09,9E+09,9E+09,9E+09]];
    TASK PERS robtarget robtPlatoonAligned:=[[2108.00,-21.16,116.06],[0.495018,-0.49502,-0.504932,-0.504932],[-1,0,-3,1],[3109,9E+09,9E+09,9E+09,9E+09,9E+09]];
    TASK PERS jointtarget jointPlatoonAligned:=[[-1.35298,49.4559,34.9342,-0.583296,-47.8646,-180.327],[3087,9E+09,9E+09,9E+09,9E+09,9E+09]];
    TASK PERS jointtarget jointPHCenterMedianLine:=[[-10.8578,-8.43553,62.8792,145.044,21.0571,31.1607],[2602,9E+09,9E+09,9E+09,9E+09,9E+09]];
    TASK PERS robtarget robtPHCenterMedianLine:=[[0,-133.7,0],[0.523896,-0.523898,-0.474903,-0.474901],[-1,1,0,0],[2602,9E+09,9E+09,9E+09,9E+09,9E+09]];
    TASK PERS jointtarget jointSHCenterMedianLine:=[[23.5615,77.3976,-15.0591,99.1075,-66.2014,-158.956],[4502,9E+09,9E+09,9E+09,9E+09,9E+09]];
    TASK PERS robtarget robtSHCenterMedianLine:=[[144.04,0,0],[0.673965,0.213937,-0.673967,-0.213939],[-1,-2,1,1],[759,9E+09,9E+09,9E+09,9E+09,9E+09]];

    TASK PERS jointtarget jointTrackHorizontal:=[[-0.987537,5.59217,51.9964,-0.824183,-94.0065,1.45921],[0,9E+09,9E+09,9E+09,9E+09,9E+09]];
    TASK PERS robtarget robtTrackHorizontal:=[[5217,215,1030],[0.5,-0.5,0.5,0.5],[-1,-1,0,1],[0,9E+09,9E+09,9E+09,9E+09,9E+09]];

    TASK PERS RecordFrameOffset rFrameOffsetSaddle{100}:=[[0,0,0,0,0,0,0,0,0],[0,0,0,0,0,0,0,0,0],[0,0,0,0,0,0,0,0,0],[0,0,0,0,0,0,0,0,0],[0,0,0,0,0,0,0,0,0],[0,0,0,0,0,0,0,0,0],[0,0,0,0,0,0,0,0,0],[0,0,0,0,0,0,0,0,0],[0,0,0,0,0,0,0,0,0],[0,0,0,0,0,0,0,0,0],[0,0,0,0,0,0,0,0,0],[0,0,0,0,0,0,0,0,0],[0,0,0,0,0,0,0,0,0],[0,0,0,0,0,0,0,0,0],[0,0,0,0,0,0,0,0,0],[0,0,0,0,0,0,0,0,0],[0,0,0,0,0,0,0,0,0],[0,0,0,0,0,0,0,0,0],[0,0,0,0,0,0,0,0,0],[0,0,0,0,0,0,0,0,0],[0,0,0,0,0,0,0,0,0],[0,0,0,0,0,0,0,0,0],[0,0,0,0,0,0,0,0,0],[0,0,0,0,0,0,0,0,0],[0,0,0,0,0,0,0,0,0],[0,0,0,0,0,0,0,0,0],[0,0,0,0,0,0,0,0,0],[0,0,0,0,0,0,0,0,0],[0,0,0,0,0,0,0,0,0],[0,0,0,0,0,0,0,0,0],[0,0,0,0,0,0,0,0,0],[0,0,0,0,0,0,0,0,0],[0,0,0,0,0,0,0,0,0],[0,0,0,0,0,0,0,0,0],[0,0,0,0,0,0,0,0,0],[0,0,0,0,0,0,0,0,0],[0,0,0,0,0,0,0,0,0],[0,0,0,0,0,0,0,0,0],[0,0,0,0,0,0,0,0,0],[0,0,0,0,0,0,0,0,0],[0,0,0,0,0,0,0,0,0],[0,0,0,0,0,0,0,0,0],[0,0,0,0,0,0,0,0,0],[0,0,0,0,0,0,0,0,0],[0,0,0,0,0,0,0,0,0],[0,0,0,0,0,0,0,0,0],[0,0,0,0,0,0,0,0,0],[0,0,0,0,0,0,0,0,0],[0,0,0,0,0,0,0,0,0],[0,0,0,0,0,0,0,0,0],[0,0,0,0,0,0,0,0,0],[0,0,0,0,0,0,0,0,0],[0,0,0,0,0,0,0,0,0],[0,0,0,0,0,0,0,0,0],[0,0,0,0,0,0,0,0,0],[0,0,0,0,0,0,0,0,0],[0,0,0,0,0,0,0,0,0],[0,0,0,0,0,0,0,0,0],[0,0,0,0,0,0,0,0,0],[0,0,0,0,0,0,0,0,0],[0,0,0,0,0,0,0,0,0],[0,0,0,0,0,0,0,0,0],[0,0,0,0,0,0,0,0,0],[0,0,0,0,0,0,0,0,0],[0,0,0,0,0,0,0,0,0],[0,0,0,0,0,0,0,0,0],[0,0,0,0,0,0,0,0,0],[0,0,0,0,0,0,0,0,0],[0,0,0,0,0,0,0,0,0],[0,0,0,0,0,0,0,0,0],[0,0,0,0,0,0,0,0,0],[0,0,0,0,0,0,0,0,0],[0,0,0,0,0,0,0,0,0],[0,0,0,0,0,0,0,0,0],[0,0,0,0,0,0,0,0,0],[0,0,0,0,0,0,0,0,0],[0,0,0,0,0,0,0,0,0],[0,0,0,0,0,0,0,0,0],[0,0,0,0,0,0,0,0,0],[0,0,0,0,0,0,0,0,0],[0,0,0,0,0,0,0,0,0],[0,0,0,0,0,0,0,0,0],[0,0,0,0,0,0,0,0,0],[0,0,0,0,0,0,0,0,0],[0,0,0,0,0,0,0,0,0],[0,0,0,0,0,0,0,0,0],[0,0,0,0,0,0,0,0,0],[0,0,0,0,0,0,0,0,0],[0,0,0,0,0,0,0,0,0],[0,0,0,0,0,0,0,0,0],[0,0,0,0,0,0,0,0,0],[0,0,0,0,0,0,0,0,0],[0,0,0,0,0,0,0,0,0],[0,0,0,0,0,0,0,0,0],[0,0,0,0,0,0,0,0,0],[0,0,0,0,0,0,0,0,0],[0,0,0,0,0,0,0,0,0],[0,0,0,0,0,0,0,0,0],[0,0,0,0,0,0,0,0,0],[0,0,0,0,0,0,0,0,0]];
    TASK PERS RecordFrameOffset rFrameOffsetPlatoon{100}:=[[0,10000,0,0,0,0,0,0,0],[0,0,0,0,0,0,0,0,0],[0,0,0,0,0,0,0,0,0],[0,0,0,0,0,0,0,0,0],[0,0,0,0,0,0,0,0,0],[0,0,0,0,0,0,0,0,0],[0,0,0,0,0,0,0,0,0],[0,0,0,0,0,0,0,0,0],[0,0,0,0,0,0,0,0,0],[0,0,0,0,0,0,0,0,0],[0,0,0,0,0,0,0,0,0],[0,0,0,0,0,0,0,0,0],[0,0,0,0,0,0,0,0,0],[0,0,0,0,0,0,0,0,0],[0,0,0,0,0,0,0,0,0],[0,0,0,0,0,0,0,0,0],[0,0,0,0,0,0,0,0,0],[0,0,0,0,0,0,0,0,0],[0,0,0,0,0,0,0,0,0],[0,0,0,0,0,0,0,0,0],[0,0,0,0,0,0,0,0,0],[0,0,0,0,0,0,0,0,0],[0,0,0,0,0,0,0,0,0],[0,0,0,0,0,0,0,0,0],[0,0,0,0,0,0,0,0,0],[0,0,0,0,0,0,0,0,0],[0,0,0,0,0,0,0,0,0],[0,0,0,0,0,0,0,0,0],[0,0,0,0,0,0,0,0,0],[0,0,0,0,0,0,0,0,0],[0,0,0,0,0,0,0,0,0],[0,0,0,0,0,0,0,0,0],[0,0,0,0,0,0,0,0,0],[0,0,0,0,0,0,0,0,0],[0,0,0,0,0,0,0,0,0],[0,0,0,0,0,0,0,0,0],[0,0,0,0,0,0,0,0,0],[0,0,0,0,0,0,0,0,0],[0,0,0,0,0,0,0,0,0],[0,0,0,0,0,0,0,0,0],[0,0,0,0,0,0,0,0,0],[0,0,0,0,0,0,0,0,0],[0,0,0,0,0,0,0,0,0],[0,0,0,0,0,0,0,0,0],[0,0,0,0,0,0,0,0,0],[0,0,0,0,0,0,0,0,0],[0,0,0,0,0,0,0,0,0],[0,0,0,0,0,0,0,0,0],[0,0,0,0,0,0,0,0,0],[0,0,0,0,0,0,0,0,0],[0,0,0,0,0,0,0,0,0],[0,0,0,0,0,0,0,0,0],[0,0,0,0,0,0,0,0,0],[0,0,0,0,0,0,0,0,0],[0,0,0,0,0,0,0,0,0],[0,0,0,0,0,0,0,0,0],[0,0,0,0,0,0,0,0,0],[0,0,0,0,0,0,0,0,0],[0,0,0,0,0,0,0,0,0],[0,0,0,0,0,0,0,0,0],[0,0,0,0,0,0,0,0,0],[0,0,0,0,0,0,0,0,0],[0,0,0,0,0,0,0,0,0],[0,0,0,0,0,0,0,0,0],[0,0,0,0,0,0,0,0,0],[0,0,0,0,0,0,0,0,0],[0,0,0,0,0,0,0,0,0],[0,0,0,0,0,0,0,0,0],[0,0,0,0,0,0,0,0,0],[0,0,0,0,0,0,0,0,0],[0,0,0,0,0,0,0,0,0],[0,0,0,0,0,0,0,0,0],[0,0,0,0,0,0,0,0,0],[0,0,0,0,0,0,0,0,0],[0,0,0,0,0,0,0,0,0],[0,0,0,0,0,0,0,0,0],[0,0,0,0,0,0,0,0,0],[0,0,0,0,0,0,0,0,0],[0,0,0,0,0,0,0,0,0],[0,0,0,0,0,0,0,0,0],[0,0,0,0,0,0,0,0,0],[0,0,0,0,0,0,0,0,0],[0,0,0,0,0,0,0,0,0],[0,0,0,0,0,0,0,0,0],[0,0,0,0,0,0,0,0,0],[0,0,0,0,0,0,0,0,0],[0,0,0,0,0,0,0,0,0],[0,0,0,0,0,0,0,0,0],[0,0,0,0,0,0,0,0,0],[0,0,0,0,0,0,0,0,0],[0,0,0,0,0,0,0,0,0],[0,0,0,0,0,0,0,0,0],[0,0,0,0,0,0,0,0,0],[0,0,0,0,0,0,0,0,0],[0,0,0,0,0,0,0,0,0],[0,0,0,0,0,0,0,0,0],[0,0,0,0,0,0,0,0,0],[0,0,0,0,0,0,0,0,0],[0,0,0,0,0,0,0,0,0],[0,0,0,0,0,0,0,0,0]];

    !*****************************************************
    !For ScanV2Module
    CONST string strRobNo:="1";
    CONST string strAiLaserName:="aiLaserScan"+strRobNo;
    CONST num numTCPLaserValue:=0;

    CONST string strScanPlatoonBranchLogFileName:="ScanPlatoonBranch"+strRobNo+".csv";
    CONST string strScanPlatoonHeaderLogFileName:="ScanPlatoonHeader"+strRobNo+".csv";
    CONST string strScanSaddleBranchLogFileName:="ScanSaddleBranch"+strRobNo+".csv";
    CONST string strScanSaddleHeaderLogFileName:="ScanSaddleHeader"+strRobNo+".csv";

    TASK PERS robtarget robtSPBLLCCenter:=[[3770,-38.1,293.7],[0.707107,-0.707107,0,0],[-1,-1,-2,1],[1447,9E+09,9E+09,9E+09,9E+09,9E+09]];
    TASK PERS robtarget robtSPBLLClosestDetect:=[[3770,-38.1,293.7],[0.5,-0.5,-0.5,-0.5],[-1,-1,-2,1],[1447,9E+09,9E+09,9E+09,9E+09,9E+09]];

    TASK PERS robtarget robtSPHLLCCenter:=[[2703.1,-133.7,0],[0.5,-0.5,0.5,0.5],[0,0,1,1],[2602,9E+09,9E+09,9E+09,9E+09,9E+09]];
    TASK PERS robtarget robtSPHLLClosestDetect:=[[2703.1,-133.7,0],[0.5,-0.5,0.5,0.5],[0,0,1,1],[2602,9E+09,9E+09,9E+09,9E+09,9E+09]];

    TASK PERS robtarget robtSSBLLCCenter:=[[955,-159.25,259.25],[3.09086E-08,3.09086E-08,-0.707107,-0.707107],[-1,-1,1,1],[4262,9E+09,9E+09,9E+09,9E+09,9E+09]];
    TASK PERS robtarget robtSSBLLClosestDetect:=[[955,-38.1,268.15],[3.09086E-08,3.09086E-08,-0.707107,-0.707107],[-1,-1,1,1],[4262,9E+09,9E+09,9E+09,9E+09,9E+09]];

    TASK PERS robtarget robtSSHLLCCenter:=[[1129.25,-159.25,0],[0.5,-0.5,-0.5,-0.5],[0,0,1,1],[4262,9E+09,9E+09,9E+09,9E+09,9E+09]];
    TASK PERS robtarget robtSSHLLClosestDetect:=[[1129.25,-108.15,0],[0.5,-0.5,-0.5,-0.5],[0,0,1,1],[4262,9E+09,9E+09,9E+09,9E+09,9E+09]];
    !*****************************************************

ENDMODULE
